REGION Network 12: Fittings - Cyle times measurement
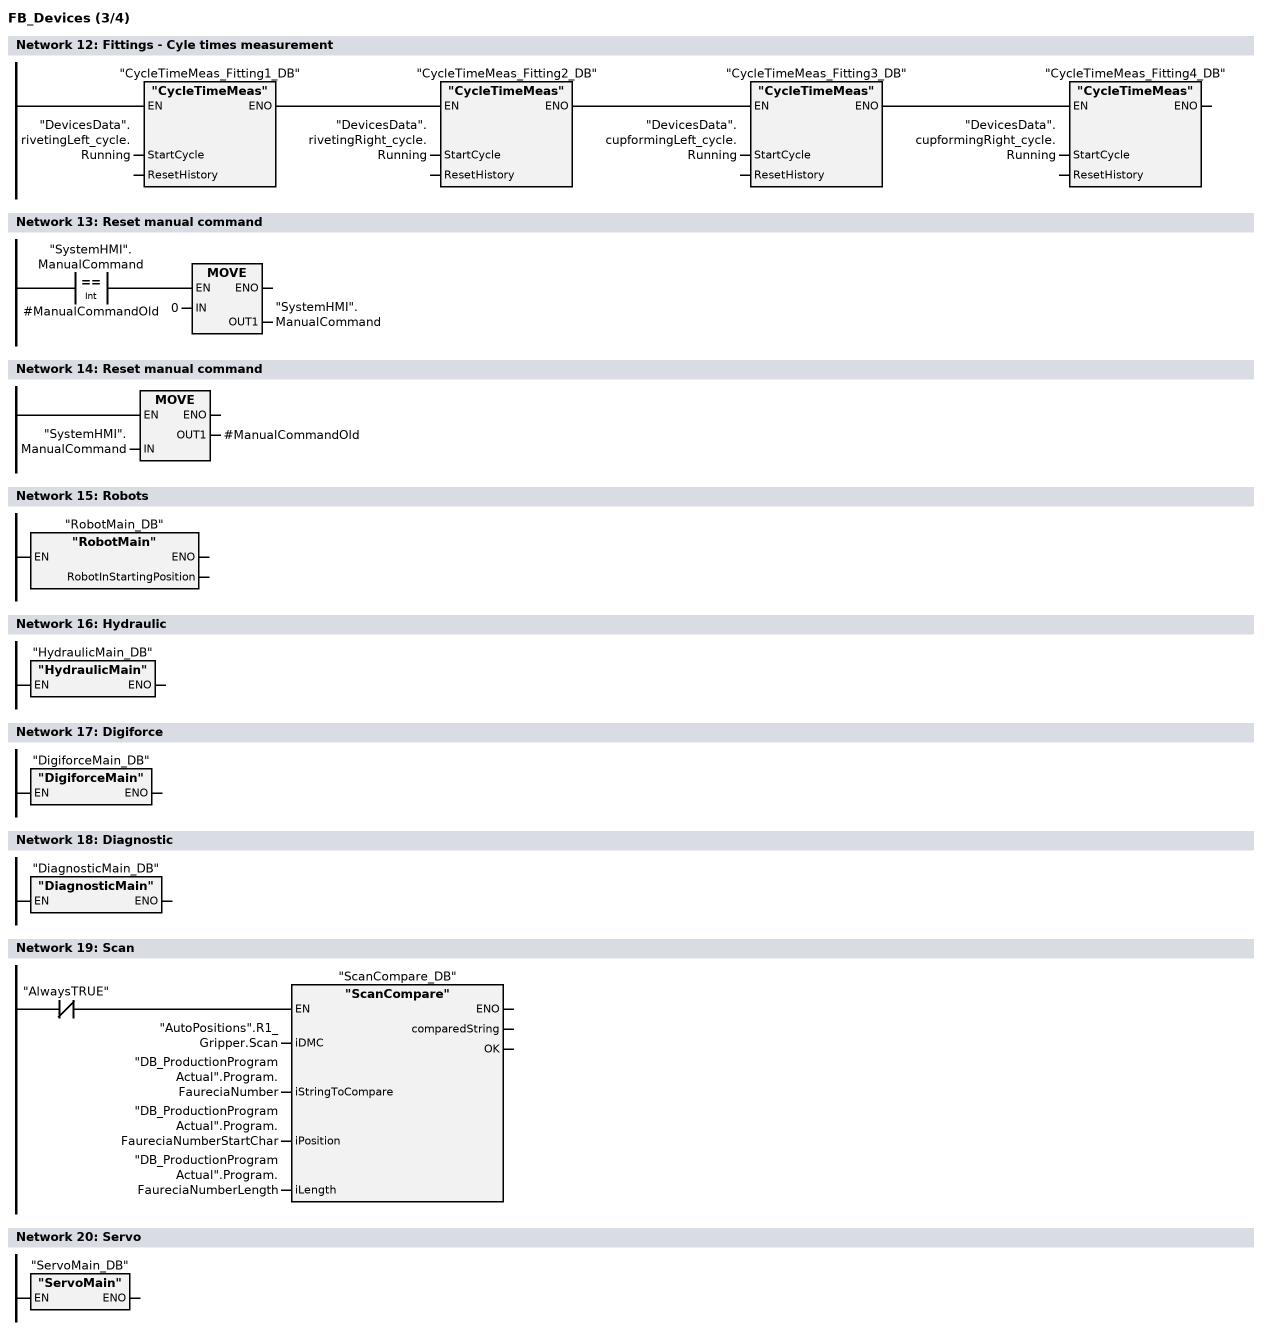
   RUNG wire#powerrail
      "CycleTimeMeas_Fitting1_DB"(StartCycle := "DevicesData".rivetingLeft_cycle.Running, ResetHistory :=)
      "CycleTimeMeas_Fitting2_DB"(StartCycle := "DevicesData".rivetingRight_cycle.Running, ResetHistory :=)
      "CycleTimeMeas_Fitting3_DB"(StartCycle := "DevicesData".cupformingLeft_cycle.Running, ResetHistory :=)
      "CycleTimeMeas_Fitting4_DB"(StartCycle := "DevicesData".cupformingRight_cycle.Running, ResetHistory :=)
   END_RUNG
   // the same network as SCL:
   "CycleTimeMeas_Fitting1_DB"(StartCycle := "DevicesData".rivetingLeft_cycle.Running, ENO => #_w1);   // "CycleTimeMeas"
   "CycleTimeMeas_Fitting2_DB"(EN := #_w1, StartCycle := "DevicesData".rivetingRight_cycle.Running, ENO => #_w2);   // "CycleTimeMeas"
   "CycleTimeMeas_Fitting3_DB"(EN := #_w2,   // "CycleTimeMeas"
                           StartCycle := "DevicesData".cupformingLeft_cycle.Running,
                           ENO => #_w3);
   IF #_w3 THEN
       "CycleTimeMeas_Fitting4_DB"(StartCycle := "DevicesData".cupformingRight_cycle.Running);   // "CycleTimeMeas"
   END_IF;
END_REGION

REGION Network 13: Reset manual command
   RUNG wire#powerrail
      { S7_Templates := "SrcType := Int" } EQ_Contact(in1 := "SystemHMI".ManualCommand, in2 := #ManualCommandOld)
      Move(in := 0, out1 => "SystemHMI".ManualCommand)
   END_RUNG
   // the same network as SCL:
   IF "SystemHMI".ManualCommand = #ManualCommandOld THEN "SystemHMI".ManualCommand := 0; END_IF;
END_REGION

REGION Network 14: Reset manual command
   RUNG wire#powerrail
      Move(in := "SystemHMI".ManualCommand, out1 => #ManualCommandOld)
   END_RUNG
   // the same network as SCL:
   #ManualCommandOld := "SystemHMI".ManualCommand;
END_REGION

REGION Network 15: Robots
   RUNG wire#powerrail
      "RobotMain_DB"(RobotInStartingPosition =>)
   END_RUNG
   // the same network as SCL:
   "RobotMain_DB"();   // "RobotMain"
END_REGION

REGION Network 16: Hydraulic
   RUNG wire#powerrail
      "HydraulicMain_DB"()
   END_RUNG
   // the same network as SCL:
   "HydraulicMain_DB"();   // "HydraulicMain"
END_REGION

REGION Network 17: Digiforce
   RUNG wire#powerrail
      "DigiforceMain_DB"()
   END_RUNG
   // the same network as SCL:
   "DigiforceMain_DB"();   // "DigiforceMain"
END_REGION

REGION Network 18: Diagnostic
   RUNG wire#powerrail
      "DiagnosticMain_DB"()
   END_RUNG
   // the same network as SCL:
   "DiagnosticMain_DB"();   // "DiagnosticMain"
END_REGION

REGION Network 19: Scan
   RUNG wire#powerrail
      I_Contact( "AlwaysTRUE" )
      "ScanCompare_DB"(iDMC := "AutoPositions".R1_Gripper.Scan, iStringToCompare := "DB_ProductionProgramActual".Program.FaureciaNumber, iPosition := "DB_ProductionProgramActual".Program.FaureciaNumberStartChar, iLength := "DB_ProductionProgramActual".Program.FaureciaNumberLength, comparedString =>, OK =>)
   END_RUNG
   // the same network as SCL:
   IF NOT "AlwaysTRUE" THEN
       "ScanCompare_DB"(iDMC := "AutoPositions".R1_Gripper.Scan,   // "ScanCompare"
                        iStringToCompare := "DB_ProductionProgramActual".Program.FaureciaNumber,
                        iPosition := "DB_ProductionProgramActual".Program.FaureciaNumberStartChar,
                        iLength := "DB_ProductionProgramActual".Program.FaureciaNumberLength);
   END_IF;
END_REGION

REGION Network 20: Servo
   RUNG wire#powerrail
      "ServoMain_DB"()
   END_RUNG
   // the same network as SCL:
   "ServoMain_DB"();   // "ServoMain"
END_REGION

REGION Network 21 (SCL): Friedrich1 R
   IF "HMIData".ManualCommand = 611 THEN
       "DevicesData".Friedrich1.Start := true;
   END_IF;

   #FriedrichUnit1_Instance(safetyOK := "safety_signals"."4L+",
                            iReady := "iRivetingReady1",
                            iZ1OK := "iRivetingZ1ok1",
                            iH1OK := "iRivetingH1ok1",
                            iH2OK := "iRivetingH2ok1",
                            iTimeOK := "iRivetingTimeOk1",
                            iNoAlarm := "iRivetingNoError1",
                            FriedrichNumber := 1,
                            Port := 39000,
                            IP1 := 192,
                            IP2 := 168,
                            IP3 := 16,
                            IP4 := 43,
                            ID := 2,
                            qStart => "qRiveting1Start",
                            qPrgbit4 => "qRiveting1Bit4",
                            qPrgbit3 => "qRiveting1Bit3",
                            qPrgbit2 => "qRiveting1Bit2",
                            qPrgbit1 => "qRiveting1Bit1",
                            qPrgbit0 => "qRiveting1Bit0",
                            RivetData := "DevicesData".Friedrich1);
   "qFriedrich1_setup_mode" := "DB_MainData".MachineMode <> 2 AND "DB_MainData".MachineMode <> 3;

   #Trig1(CLK:="DevicesData".Friedrich1.OK);
   #Trig2(CLK:="DevicesData".Friedrich1.NOK);
   "RivetingHistoryRight_DB"(iNewCycle := #Trig1.Q OR #Trig2.Q,
                             iData := "DevicesData".Friedrich1);

   #RivetingCycleRight_Instance(parameters := "DB_ProductionProgramActual".Program.Riveting_program_right,
                                basicPosition := "DevicesData".Friedrich1.Ready AND "DevicesData".Cylinders[MM340_RivetingUnitRight].InBp AND "DevicesData".Cylinders[MM344_RivetingSupportRight].InBp,
                                twoRivets := "DB_ProductionProgramActual".Program.Total_number_of_rivets_4,
                                MeasuredData1=>"AutoInfo".PartMeasuredData.RightRiveting1,
                                MeasuredData2=>"AutoInfo".PartMeasuredData.RightRiveting2,
                                riveter := "DevicesData".Friedrich1,
                                data := "DevicesData".rivetingRight_cycle,
                                cylinderSupport := "DevicesData".Cylinders[MM344_RivetingSupportRight],
                                cylinderShift := "DevicesData".Cylinders[MM340_RivetingUnitRight]);
END_REGION

REGION Network 22 (SCL): Friedrich2 L
   IF "HMIData".ManualCommand = 612 THEN
       "DevicesData".Friedrich2.Start := true;
   END_IF;
   #FriedrichUnit2_Instance(safetyOK := "safety_signals"."4L+",
                            iReady := "iRivetingReady2",
                            iZ1OK := "iRivetingZ1ok2",
                            iH1OK := "iRivetingH1ok2",
                            iH2OK := "iRivetingH2ok2",
                            iTimeOK := "iRivetingTimeOk2",
                            iNoAlarm := "iRivetingNoError2",
                            FriedrichNumber := 2,
                            Port := 39000,
                            IP1 := 192,
                            IP2 := 168,
                            IP3 := 16,
                            IP4 := 44,
                            ID := 3,
                            qStart => "qRiveting2Start",
                            qPrgbit4 => "qRiveting2Bit4",
                            qPrgbit3 => "qRiveting2Bit3",
                            qPrgbit2 => "qRiveting2Bit2",
                            qPrgbit1 => "qRiveting2Bit1",
                            qPrgbit0 => "qRiveting2Bit0",
                            RivetData := "DevicesData".Friedrich2);
   "qFriedrich2_setup_mode" := "DB_MainData".MachineMode <> 2 AND "DB_MainData".MachineMode <> 3;

   #Trig3(CLK:="DevicesData".Friedrich2.OK);
   #Trig4(CLK:="DevicesData".Friedrich2.NOK);
   "RivetingHistoryLeft_DB"(iNewCycle := #Trig3.Q OR #Trig4.Q,
                            iData := "DevicesData".Friedrich2);

   #RivetingCycleLeft_Instance(parameters := "DB_ProductionProgramActual".Program.Riveting_program_left,
                               basicPosition := "DevicesData".Friedrich2.Ready AND "DevicesData".Cylinders[MM342_RivetingUnitLeft].InBp AND "DevicesData".Cylinders[MM346_RivetingSupportLeft].InBp,
                               twoRivets := "DB_ProductionProgramActual".Program.Total_number_of_rivets_4,
                               MeasuredData1=>"AutoInfo".PartMeasuredData.LeftRiveting1,
                               MeasuredData2=>"AutoInfo".PartMeasuredData.LeftRiveting2,
                               riveter := "DevicesData".Friedrich2,
                               data := "DevicesData".rivetingLeft_cycle,
                               cylinderSupport := "DevicesData".Cylinders[MM346_RivetingSupportLeft],
                               cylinderShift := "DevicesData".Cylinders[MM342_RivetingUnitLeft]);

   REGION cycles handshake
       IF "SystemHMI".AutomaticMode THEN
           IF "DevicesData".cupformingLeft_cycle.Done AND "DevicesData".cupformingRight_cycle.Done THEN
               "DevicesData".rivetingLeft_cycle.ContinueFitting := TRUE;
               "DevicesData".rivetingRight_cycle.ContinueFitting := TRUE;
           END_IF;
       END_IF;
       "DevicesData".rivetingLeft_cycle.ContinueFitting := TRUE;
       "DevicesData".rivetingRight_cycle.ContinueFitting := TRUE;

       IF "SystemHMI".ManualMode THEN
           "DevicesData".rivetingLeft_cycle.ContinueFitting := true;
           "DevicesData".rivetingRight_cycle.ContinueFitting := true;
       END_IF;
   END_REGION
END_REGION

REGION Network 23
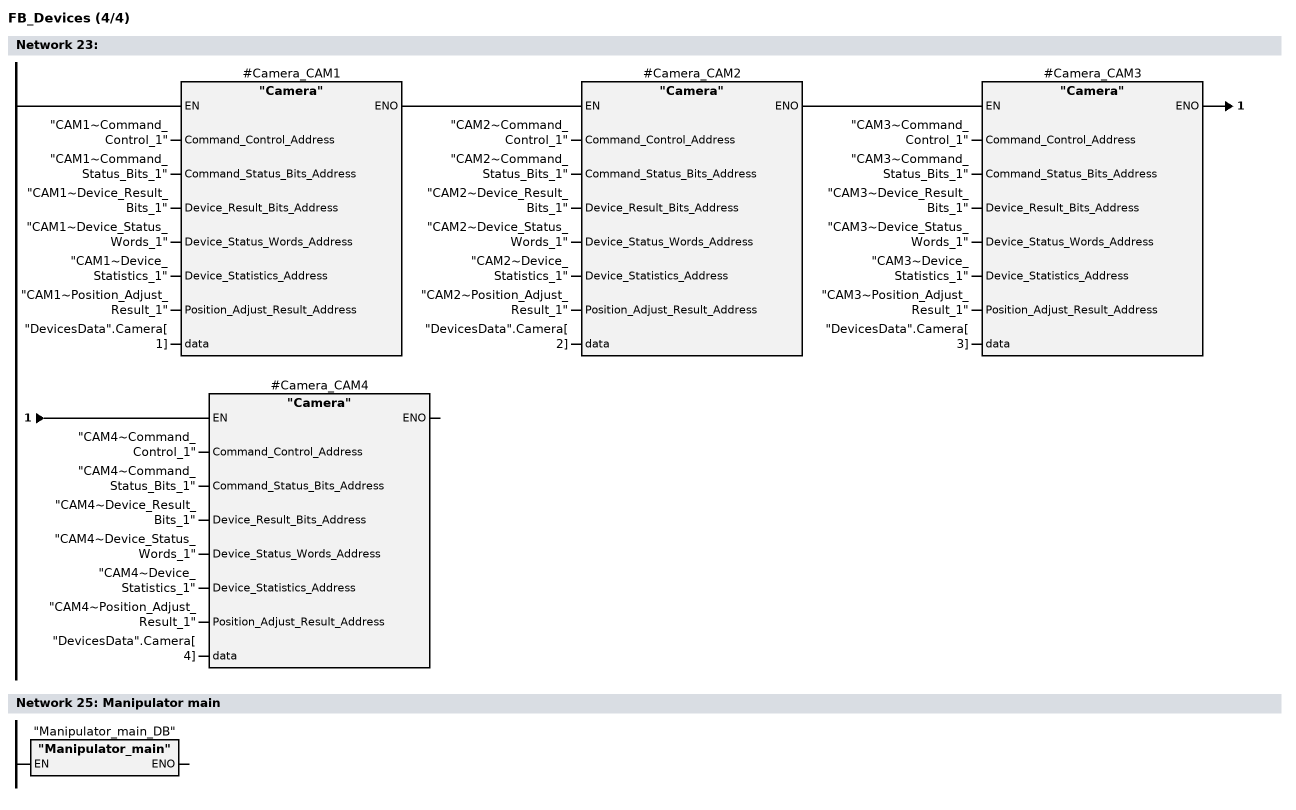
   RUNG wire#powerrail
      #Camera_CAM1(Command_Control_Address := "CAM1~Command_Control_1", Command_Status_Bits_Address := "CAM1~Command_Status_Bits_1", Device_Result_Bits_Address := "CAM1~Device_Result_Bits_1", Device_Status_Words_Address := "CAM1~Device_Status_Words_1", Device_Statistics_Address := "CAM1~Device_Statistics_1", Position_Adjust_Result_Address := "CAM1~Position_Adjust_Result_1", data := "DevicesData".Camera[1])
      #Camera_CAM2(Command_Control_Address := "CAM2~Command_Control_1", Command_Status_Bits_Address := "CAM2~Command_Status_Bits_1", Device_Result_Bits_Address := "CAM2~Device_Result_Bits_1", Device_Status_Words_Address := "CAM2~Device_Status_Words_1", Device_Statistics_Address := "CAM2~Device_Statistics_1", Position_Adjust_Result_Address := "CAM2~Position_Adjust_Result_1", data := "DevicesData".Camera[2])
      #Camera_CAM3(Command_Control_Address := "CAM3~Command_Control_1", Command_Status_Bits_Address := "CAM3~Command_Status_Bits_1", Device_Result_Bits_Address := "CAM3~Device_Result_Bits_1", Device_Status_Words_Address := "CAM3~Device_Status_Words_1", Device_Statistics_Address := "CAM3~Device_Statistics_1", Position_Adjust_Result_Address := "CAM3~Position_Adjust_Result_1", data := "DevicesData".Camera[3])
      #Camera_CAM4(Command_Control_Address := "CAM4~Command_Control_1", Command_Status_Bits_Address := "CAM4~Command_Status_Bits_1", Device_Result_Bits_Address := "CAM4~Device_Result_Bits_1", Device_Status_Words_Address := "CAM4~Device_Status_Words_1", Device_Statistics_Address := "CAM4~Device_Statistics_1", Position_Adjust_Result_Address := "CAM4~Position_Adjust_Result_1", data := "DevicesData".Camera[4])
   END_RUNG
   // the same network as SCL:
   #Camera_CAM1(Command_Control_Address := "CAM1~Command_Control_1",   // "Camera"
                Command_Status_Bits_Address := "CAM1~Command_Status_Bits_1",
                Device_Result_Bits_Address := "CAM1~Device_Result_Bits_1",
                Device_Status_Words_Address := "CAM1~Device_Status_Words_1",
                Device_Statistics_Address := "CAM1~Device_Statistics_1",
                Position_Adjust_Result_Address := "CAM1~Position_Adjust_Result_1",
                data := "DevicesData".Camera[1],
                ENO => #_w1);
   #Camera_CAM2(EN := #_w1,   // "Camera"
                Command_Control_Address := "CAM2~Command_Control_1",
                Command_Status_Bits_Address := "CAM2~Command_Status_Bits_1",
                Device_Result_Bits_Address := "CAM2~Device_Result_Bits_1",
                Device_Status_Words_Address := "CAM2~Device_Status_Words_1",
                Device_Statistics_Address := "CAM2~Device_Statistics_1",
                Position_Adjust_Result_Address := "CAM2~Position_Adjust_Result_1",
                data := "DevicesData".Camera[2],
                ENO => #_w2);
   #Camera_CAM3(EN := #_w2,   // "Camera"
                Command_Control_Address := "CAM3~Command_Control_1",
                Command_Status_Bits_Address := "CAM3~Command_Status_Bits_1",
                Device_Result_Bits_Address := "CAM3~Device_Result_Bits_1",
                Device_Status_Words_Address := "CAM3~Device_Status_Words_1",
                Device_Statistics_Address := "CAM3~Device_Statistics_1",
                Position_Adjust_Result_Address := "CAM3~Position_Adjust_Result_1",
                data := "DevicesData".Camera[3],
                ENO => #_w3);
   IF #_w3 THEN
       #Camera_CAM4(Command_Control_Address := "CAM4~Command_Control_1",   // "Camera"
                    Command_Status_Bits_Address := "CAM4~Command_Status_Bits_1",
                    Device_Result_Bits_Address := "CAM4~Device_Result_Bits_1",
                    Device_Status_Words_Address := "CAM4~Device_Status_Words_1",
                    Device_Statistics_Address := "CAM4~Device_Statistics_1",
                    Position_Adjust_Result_Address := "CAM4~Position_Adjust_Result_1",
                    data := "DevicesData".Camera[4]);
   END_IF;
END_REGION

REGION Network 24 (SCL)
   "DevicesData".Camera[1].ProgramNumber := USINT_TO_SINT("DB_ProductionProgramActual".Program.Camera_program[1]);
   "DevicesData".Camera[2].ProgramNumber := USINT_TO_SINT("DB_ProductionProgramActual".Program.Camera_program[2]);
   "DevicesData".Camera[3].ProgramNumber := USINT_TO_SINT("DB_ProductionProgramActual".Program.Camera_program[3]);
   "DevicesData".Camera[4].ProgramNumber := USINT_TO_SINT("DB_ProductionProgramActual".Program.Camera_program[4]);
END_REGION

REGION Network 25: Manipulator main
   RUNG wire#powerrail
      "Manipulator_main_DB"()
   END_RUNG
   // the same network as SCL:
   "Manipulator_main_DB"();   // "Manipulator_main"
END_REGION

REGION Network 26: Readers
END_REGION
END_FUNCTION_BLOCK

FUNCTION_BLOCK "CylindersMain"
{ S7_Optimized_Access := 'TRUE' }
VERSION : 0.1
   VAR 
      res : Bool;
   END_VAR


BEGIN
	
	"CylinderGeneratedCalls_DB"();
	
	"CylinderCollisions"();
	
	"CylindersHMIMessage"(CylinderNumber=>"CylindersHMI".CylinderInfoHMI,
	                      CylinderAction=>"CylindersHMI".CylinderInfoHMIAction);
	
END_FUNCTION_BLOCK

FUNCTION_BLOCK "FB_TurnTable"   // FB3600, LAD
{ S7_Optimized_Access := 'TRUE' }
VERSION : 0.1
// stored: AutoNumber false, IsIECCheckEnabled false, IsRetainMemResEnabled false, MemoryReserve 100, SetENOAutomatically false, UDAEnableTagReadback false
   VAR_INPUT
      iTurnTableInputs : Word;
      iPower : Bool;
      iSafety : Bool;
      iReset : Bool;
      iErrorReset : Bool;
      iManualMode : Bool;
      iAutomaticMode : Bool;
      iTurnTableInSafetyPosition : Bool;
   END_VAR
   VAR_OUTPUT
      qTurnTableOutputs : Word;
      qeCommunication : Bool;
      qeTurnTablePosition : Bool;
      qeTurnTableSafetyPosition : Bool;
      qeTimeout : Bool;
      qePositionRunOver : Bool;
      qeSafety : Bool;
      qeSumError : Bool;
      qeSumWarning : Bool;
   END_VAR
   VAR_IN_OUT
      iqTurnTable : "UDT_TurnTable";
   END_VAR
   VAR
      Edges : Struct
         Enabled : Bool;
         IndexerInPosition : Bool;
      END_STRUCT;
      TONs : Struct
         tDelayCommunication : TON_TIME;
         tDelayPositionError { S7_SetPoint := 'True'} : TON_TIME;
         tDelayErrorReset { S7_SetPoint := 'True'} : TON_TIME;
      END_STRUCT;
   END_VAR
   VAR RETAIN
      RetentiveData : Struct
         LastDirection : Bool;
      END_STRUCT;
   END_VAR
   VAR
      Commands : "UDT_TurnTableCommands";
   END_VAR
   VAR_TEMP
      mode_status : Struct
         manual_mode : Bool;
         automatic_mode : Bool;
         mode_active : Bool;
      END_STRUCT;
      bit : Bool;
      error : Bool;
      ready_to_cw : Bool;
      ready_to_ccw : Bool;
      ready_to_jog : Bool;
      ready_to_start : Bool;
   END_VAR
   VAR_TEMP   // added for the SCL form of the ladder/FBD networks
      _w1 : Bool;
      _w2 : Bool;
      _w3 : Bool;
   END_VAR
BEGIN

REGION Network 1: Read inputs
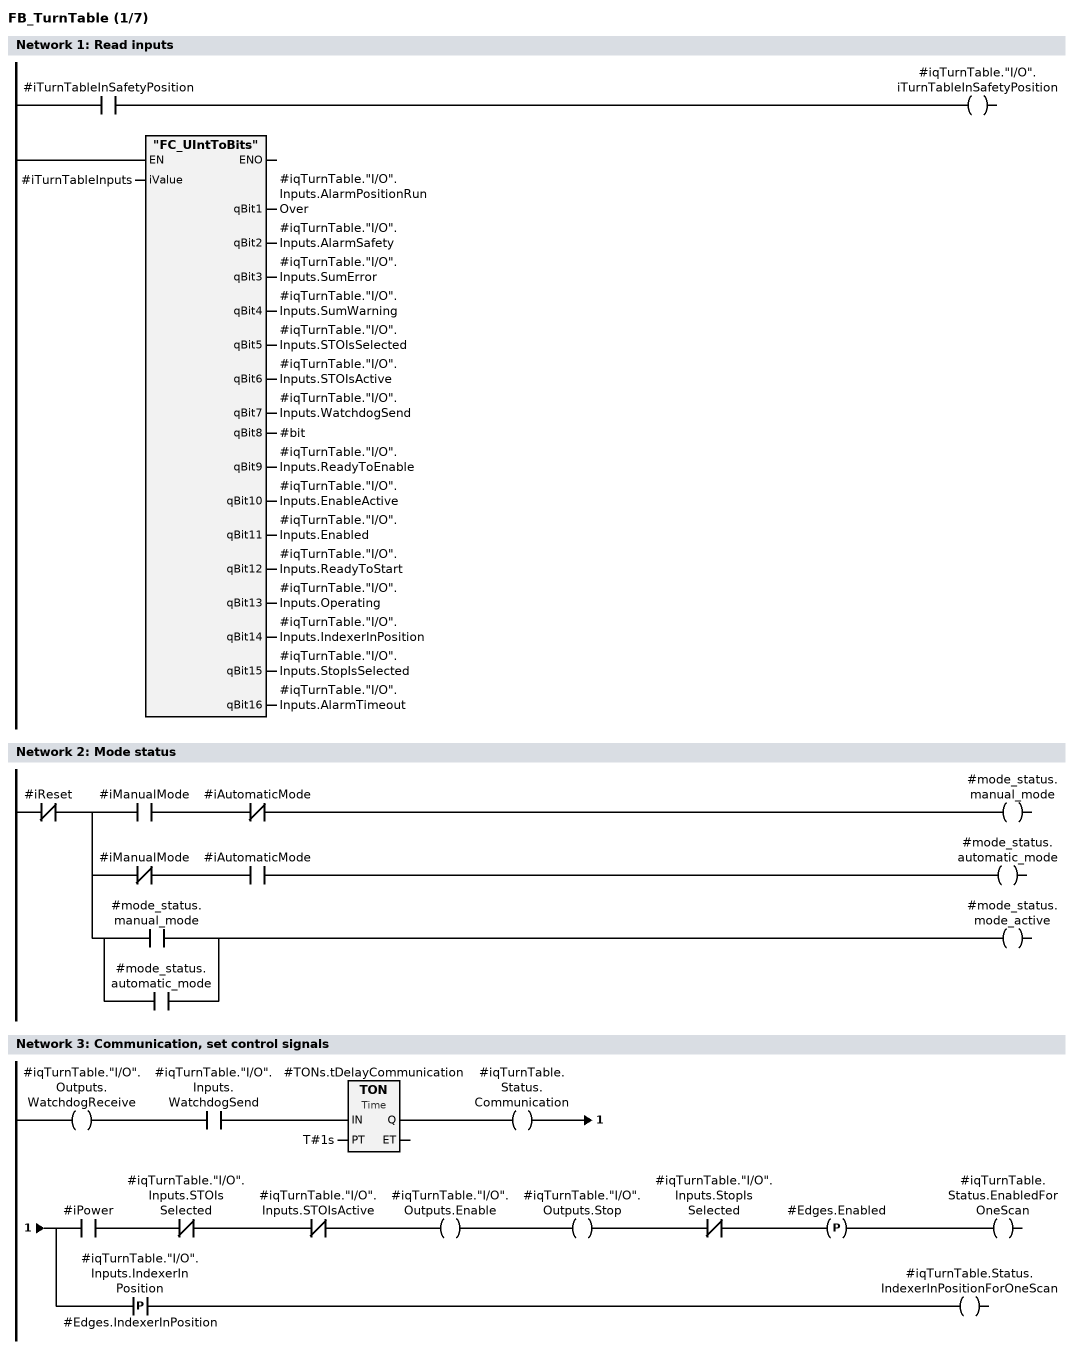
   RUNG wire#powerrail
      Contact( #iTurnTableInSafetyPosition )
      Coil( #iqTurnTable."I/O".iTurnTableInSafetyPosition )
   END_RUNG
   RUNG wire#powerrail
      "FC_UIntToBits"(iValue := #iTurnTableInputs, qBit1 => #iqTurnTable."I/O".Inputs.AlarmPositionRunOver, qBit2 => #iqTurnTable."I/O".Inputs.AlarmSafety, qBit3 => #iqTurnTable."I/O".Inputs.SumError, qBit4 => #iqTurnTable."I/O".Inputs.SumWarning, qBit5 => #iqTurnTable."I/O".Inputs.STOIsSelected, qBit6 => #iqTurnTable."I/O".Inputs.STOIsActive, qBit7 => #iqTurnTable."I/O".Inputs.WatchdogSend, qBit8 => #bit, qBit9 => #iqTurnTable."I/O".Inputs.ReadyToEnable, qBit10 => #iqTurnTable."I/O".Inputs.EnableActive, qBit11 => #iqTurnTable."I/O".Inputs.Enabled, qBit12 => #iqTurnTable."I/O".Inputs.ReadyToStart, qBit13 => #iqTurnTable."I/O".Inputs.Operating, qBit14 => #iqTurnTable."I/O".Inputs.IndexerInPosition, qBit15 => #iqTurnTable."I/O".Inputs.StopIsSelected, qBit16 => #iqTurnTable."I/O".Inputs.AlarmTimeout)
   END_RUNG
   // the same network as SCL:
   #iqTurnTable."I/O".iTurnTableInSafetyPosition := #iTurnTableInSafetyPosition;
   "FC_UIntToBits"(iValue := #iTurnTableInputs,
                   qBit1 => #iqTurnTable."I/O".Inputs.AlarmPositionRunOver,
                   qBit2 => #iqTurnTable."I/O".Inputs.AlarmSafety,
                   qBit3 => #iqTurnTable."I/O".Inputs.SumError,
                   qBit4 => #iqTurnTable."I/O".Inputs.SumWarning,
                   qBit5 => #iqTurnTable."I/O".Inputs.STOIsSelected,
                   qBit6 => #iqTurnTable."I/O".Inputs.STOIsActive,
                   qBit7 => #iqTurnTable."I/O".Inputs.WatchdogSend,
                   qBit8 => #bit,
                   qBit9 => #iqTurnTable."I/O".Inputs.ReadyToEnable,
                   qBit10 => #iqTurnTable."I/O".Inputs.EnableActive,
                   qBit11 => #iqTurnTable."I/O".Inputs.Enabled,
                   qBit12 => #iqTurnTable."I/O".Inputs.ReadyToStart,
                   qBit13 => #iqTurnTable."I/O".Inputs.Operating,
                   qBit14 => #iqTurnTable."I/O".Inputs.IndexerInPosition,
                   qBit15 => #iqTurnTable."I/O".Inputs.StopIsSelected,
                   qBit16 => #iqTurnTable."I/O".Inputs.AlarmTimeout);
END_REGION

REGION Network 2: Mode status
   RUNG wire#powerrail
      I_Contact( #iReset )
      wire#w1
      Contact( #iManualMode )
      I_Contact( #iAutomaticMode )
      Coil( #mode_status.manual_mode )
   END_RUNG
   RUNG wire#w1
      I_Contact( #iManualMode )
      Contact( #iAutomaticMode )
      Coil( #mode_status.automatic_mode )
   END_RUNG
   RUNG wire#w1
      Contact( #mode_status.manual_mode )
      wire#w2
      Coil( #mode_status.mode_active )
   END_RUNG
   RUNG wire#w1
      Contact( #mode_status.automatic_mode )
   END_RUNG wire#w2
   // the same network as SCL:
   #mode_status.manual_mode := NOT #iReset AND #iManualMode AND NOT #iAutomaticMode;
   #mode_status.automatic_mode := NOT #iReset AND NOT #iManualMode AND #iAutomaticMode;
   #mode_status.mode_active := NOT #iReset AND (#mode_status.manual_mode OR #mode_status.automatic_mode);
END_REGION

REGION Network 3: Communication, set control signals
   RUNG wire#powerrail
      Coil( #iqTurnTable."I/O".Outputs.WatchdogReceive )
      Contact( #iqTurnTable."I/O".Inputs.WatchdogSend )
      { S7_Templates := "time_type := Time" } #TONs.tDelayCommunication.TON(pt := T#1s, et =>)
      Coil( #iqTurnTable.Status.Communication )
      wire#w1
      Contact( #iPower )
      I_Contact( #iqTurnTable."I/O".Inputs.STOIsSelected )
      I_Contact( #iqTurnTable."I/O".Inputs.STOIsActive )
      Coil( #iqTurnTable."I/O".Outputs.Enable )
      Coil( #iqTurnTable."I/O".Outputs.Stop )
      I_Contact( #iqTurnTable."I/O".Inputs.StopIsSelected )
      P_Trig( #Edges.Enabled )
      Coil( #iqTurnTable.Status.EnabledForOneScan )
   END_RUNG
   RUNG wire#w1
      P_Contact(operand := #iqTurnTable."I/O".Inputs.IndexerInPosition, bit := #Edges.IndexerInPosition)
      Coil( #iqTurnTable.Status.IndexerInPositionForOneScan )
   END_RUNG
   // the same network as SCL:
   #iqTurnTable."I/O".Outputs.WatchdogReceive := TRUE;
   #TONs.tDelayCommunication.TON(IN := #iqTurnTable."I/O".Inputs.WatchdogSend, PT := T#1s);
   #iqTurnTable.Status.Communication := #TONs.tDelayCommunication.Q;
   #iqTurnTable."I/O".Outputs.Enable := #TONs.tDelayCommunication.Q AND #iPower AND NOT #iqTurnTable."I/O".Inputs.STOIsSelected AND NOT #iqTurnTable."I/O".Inputs.STOIsActive;
   #iqTurnTable."I/O".Outputs.Stop := #iqTurnTable."I/O".Outputs.Enable;
   #_w1 := #iqTurnTable."I/O".Outputs.Enable AND NOT #iqTurnTable."I/O".Inputs.StopIsSelected;
   #_w2 := #_w1 AND NOT #Edges.Enabled;   // rising edge
   #Edges.Enabled := #_w1;
   #iqTurnTable.Status.EnabledForOneScan := #_w2;
   #_w3 := #TONs.tDelayCommunication.Q AND #iqTurnTable."I/O".Inputs.IndexerInPosition AND NOT #Edges.IndexerInPosition;   // rising edge of #iqTurnTable."I/O".Inputs.IndexerInPosition
   #Edges.IndexerInPosition := #iqTurnTable."I/O".Inputs.IndexerInPosition;
   #iqTurnTable.Status.IndexerInPositionForOneScan := #_w3;
END_REGION

REGION Network 4: Errors
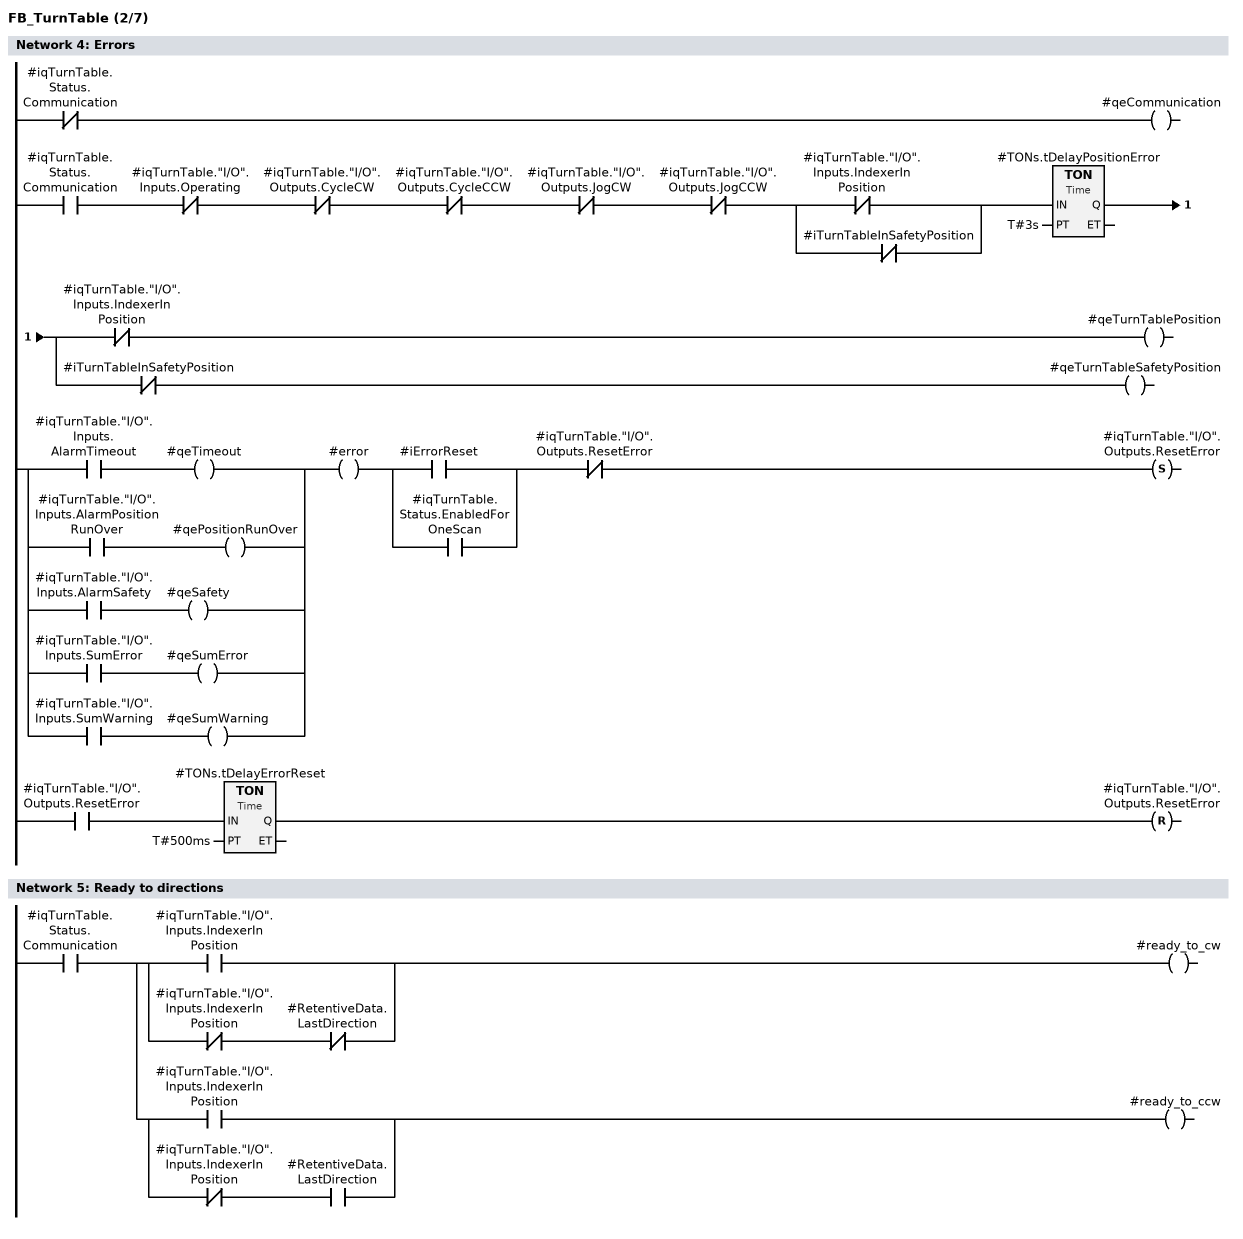
   RUNG wire#powerrail
      I_Contact( #iqTurnTable.Status.Communication )
      Coil( #qeCommunication )
   END_RUNG
   RUNG wire#powerrail
      Contact( #iqTurnTable.Status.Communication )
      I_Contact( #iqTurnTable."I/O".Inputs.Operating )
      I_Contact( #iqTurnTable."I/O".Outputs.CycleCW )
      I_Contact( #iqTurnTable."I/O".Outputs.CycleCCW )
      I_Contact( #iqTurnTable."I/O".Outputs.JogCW )
      I_Contact( #iqTurnTable."I/O".Outputs.JogCCW )
      wire#w1
      I_Contact( #iqTurnTable."I/O".Inputs.IndexerInPosition )
      wire#w2
      { S7_Templates := "time_type := Time" } #TONs.tDelayPositionError.TON(pt := T#3s, et =>)
      wire#w3
      I_Contact( #iqTurnTable."I/O".Inputs.IndexerInPosition )
      Coil( #qeTurnTablePosition )
   END_RUNG
   RUNG wire#w1
      I_Contact( #iTurnTableInSafetyPosition )
   END_RUNG wire#w2
   RUNG wire#w3
      I_Contact( #iTurnTableInSafetyPosition )
      Coil( #qeTurnTableSafetyPosition )
   END_RUNG
   RUNG wire#powerrail
      Contact( #iqTurnTable."I/O".Inputs.AlarmTimeout )
      Coil( #qeTimeout )
      wire#w4
      Coil( #error )
      wire#w5
      Contact( #iErrorReset )
      wire#w6
      I_Contact( #iqTurnTable."I/O".Outputs.ResetError )
      S_Coil( #iqTurnTable."I/O".Outputs.ResetError )
   END_RUNG
   RUNG wire#powerrail
      Contact( #iqTurnTable."I/O".Inputs.AlarmPositionRunOver )
      Coil( #qePositionRunOver )
   END_RUNG wire#w4
   RUNG wire#powerrail
      Contact( #iqTurnTable."I/O".Inputs.AlarmSafety )
      Coil( #qeSafety )
   END_RUNG wire#w4
   RUNG wire#powerrail
      Contact( #iqTurnTable."I/O".Inputs.SumError )
      Coil( #qeSumError )
   END_RUNG wire#w4
   RUNG wire#powerrail
      Contact( #iqTurnTable."I/O".Inputs.SumWarning )
      Coil( #qeSumWarning )
   END_RUNG wire#w4
   RUNG wire#w5
      Contact( #iqTurnTable.Status.EnabledForOneScan )
   END_RUNG wire#w6
   RUNG wire#powerrail
      Contact( #iqTurnTable."I/O".Outputs.ResetError )
      { S7_Templates := "time_type := Time" } #TONs.tDelayErrorReset.TON(pt := T#500ms, et =>)
      R_Coil( #iqTurnTable."I/O".Outputs.ResetError )
   END_RUNG
   // the same network as SCL:
   #qeCommunication := NOT #iqTurnTable.Status.Communication;
   #TONs.tDelayPositionError.TON(IN := #iqTurnTable.Status.Communication AND NOT #iqTurnTable."I/O".Inputs.Operating AND NOT #iqTurnTable."I/O".Outputs.CycleCW AND NOT #iqTurnTable."I/O".Outputs.CycleCCW AND NOT #iqTurnTable."I/O".Outputs.JogCW AND NOT #iqTurnTable."I/O".Outputs.JogCCW AND (NOT #iqTurnTable."I/O".Inputs.IndexerInPosition OR NOT #iTurnTableInSafetyPosition),
                           PT := T#3s);
   #qeTurnTablePosition := #TONs.tDelayPositionError.Q AND NOT #iqTurnTable."I/O".Inputs.IndexerInPosition;
   #qeTurnTableSafetyPosition := #TONs.tDelayPositionError.Q AND NOT #iTurnTableInSafetyPosition;
   #qeTimeout := #iqTurnTable."I/O".Inputs.AlarmTimeout;
   #qePositionRunOver := #iqTurnTable."I/O".Inputs.AlarmPositionRunOver;
   #qeSafety := #iqTurnTable."I/O".Inputs.AlarmSafety;
   #qeSumError := #iqTurnTable."I/O".Inputs.SumError;
   #qeSumWarning := #iqTurnTable."I/O".Inputs.SumWarning;
   #error := #iqTurnTable."I/O".Inputs.AlarmTimeout OR #iqTurnTable."I/O".Inputs.AlarmPositionRunOver OR #iqTurnTable."I/O".Inputs.AlarmSafety OR #iqTurnTable."I/O".Inputs.SumError OR #iqTurnTable."I/O".Inputs.SumWarning;
   IF #error AND (#iErrorReset OR #iqTurnTable.Status.EnabledForOneScan) AND NOT #iqTurnTable."I/O".Outputs.ResetError THEN
       #iqTurnTable."I/O".Outputs.ResetError := TRUE;
   END_IF;
   #TONs.tDelayErrorReset.TON(IN := #iqTurnTable."I/O".Outputs.ResetError, PT := T#500ms);
   IF #TONs.tDelayErrorReset.Q THEN #iqTurnTable."I/O".Outputs.ResetError := FALSE; END_IF;
END_REGION

REGION Network 5: Ready to directions
   RUNG wire#powerrail
      Contact( #iqTurnTable.Status.Communication )
      wire#w1
      Contact( #iqTurnTable."I/O".Inputs.IndexerInPosition )
      wire#w2
      Coil( #ready_to_cw )
   END_RUNG
   RUNG wire#w1
      I_Contact( #iqTurnTable."I/O".Inputs.IndexerInPosition )
      I_Contact( #RetentiveData.LastDirection )
   END_RUNG wire#w2
   RUNG wire#w1
      Contact( #iqTurnTable."I/O".Inputs.IndexerInPosition )
      wire#w3
      Coil( #ready_to_ccw )
   END_RUNG
   RUNG wire#w1
      I_Contact( #iqTurnTable."I/O".Inputs.IndexerInPosition )
      Contact( #RetentiveData.LastDirection )
   END_RUNG wire#w3
   // the same network as SCL:
   #ready_to_cw := #iqTurnTable.Status.Communication AND (#iqTurnTable."I/O".Inputs.IndexerInPosition OR (NOT #iqTurnTable."I/O".Inputs.IndexerInPosition AND NOT #RetentiveData.LastDirection));
   #ready_to_ccw := #iqTurnTable.Status.Communication AND (#iqTurnTable."I/O".Inputs.IndexerInPosition OR (NOT #iqTurnTable."I/O".Inputs.IndexerInPosition AND #RetentiveData.LastDirection));
END_REGION

REGION Network 6: Ready to jog
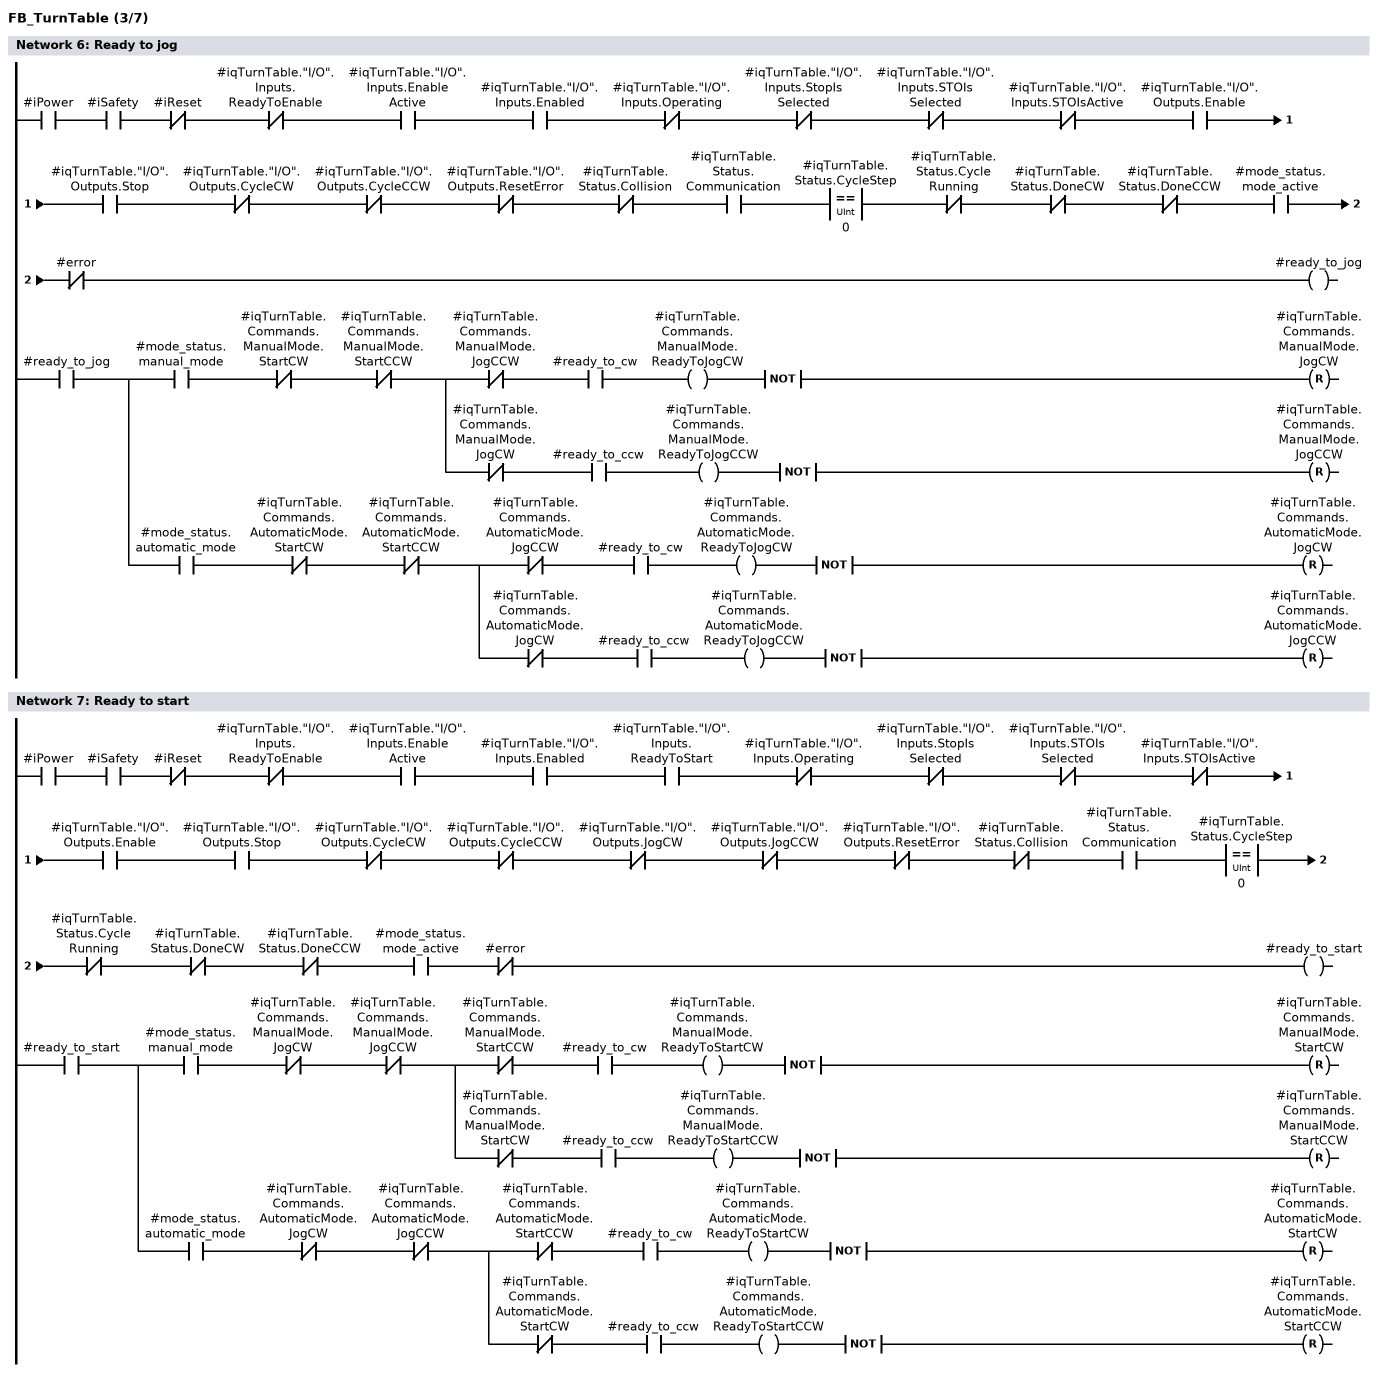
   RUNG wire#powerrail
      Contact( #iPower )
      Contact( #iSafety )
      I_Contact( #iReset )
      I_Contact( #iqTurnTable."I/O".Inputs.ReadyToEnable )
      Contact( #iqTurnTable."I/O".Inputs.EnableActive )
      Contact( #iqTurnTable."I/O".Inputs.Enabled )
      I_Contact( #iqTurnTable."I/O".Inputs.Operating )
      I_Contact( #iqTurnTable."I/O".Inputs.StopIsSelected )
      I_Contact( #iqTurnTable."I/O".Inputs.STOIsSelected )
      I_Contact( #iqTurnTable."I/O".Inputs.STOIsActive )
      Contact( #iqTurnTable."I/O".Outputs.Enable )
      Contact( #iqTurnTable."I/O".Outputs.Stop )
      I_Contact( #iqTurnTable."I/O".Outputs.CycleCW )
      I_Contact( #iqTurnTable."I/O".Outputs.CycleCCW )
      I_Contact( #iqTurnTable."I/O".Outputs.ResetError )
      I_Contact( #iqTurnTable.Status.Collision )
      Contact( #iqTurnTable.Status.Communication )
      { S7_Templates := "SrcType := UInt" } EQ_Contact(in1 := #iqTurnTable.Status.CycleStep, in2 := 0)
      I_Contact( #iqTurnTable.Status.CycleRunning )
      I_Contact( #iqTurnTable.Status.DoneCW )
      I_Contact( #iqTurnTable.Status.DoneCCW )
      Contact( #mode_status.mode_active )
      I_Contact( #error )
      Coil( #ready_to_jog )
   END_RUNG
   RUNG wire#powerrail
      Contact( #ready_to_jog )
      wire#w1
      Contact( #mode_status.manual_mode )
      I_Contact( #iqTurnTable.Commands.ManualMode.StartCW )
      I_Contact( #iqTurnTable.Commands.ManualMode.StartCCW )
      wire#w2
      I_Contact( #iqTurnTable.Commands.ManualMode.JogCCW )
      Contact( #ready_to_cw )
      Coil( #iqTurnTable.Commands.ManualMode.ReadyToJogCW )
      Not()
      R_Coil( #iqTurnTable.Commands.ManualMode.JogCW )
   END_RUNG
   RUNG wire#w2
      I_Contact( #iqTurnTable.Commands.ManualMode.JogCW )
      Contact( #ready_to_ccw )
      Coil( #iqTurnTable.Commands.ManualMode.ReadyToJogCCW )
      Not()
      R_Coil( #iqTurnTable.Commands.ManualMode.JogCCW )
   END_RUNG
   RUNG wire#w1
      Contact( #mode_status.automatic_mode )
      I_Contact( #iqTurnTable.Commands.AutomaticMode.StartCW )
      I_Contact( #iqTurnTable.Commands.AutomaticMode.StartCCW )
      wire#w3
      I_Contact( #iqTurnTable.Commands.AutomaticMode.JogCCW )
      Contact( #ready_to_cw )
      Coil( #iqTurnTable.Commands.AutomaticMode.ReadyToJogCW )
      Not()
      R_Coil( #iqTurnTable.Commands.AutomaticMode.JogCW )
   END_RUNG
   RUNG wire#w3
      I_Contact( #iqTurnTable.Commands.AutomaticMode.JogCW )
      Contact( #ready_to_ccw )
      Coil( #iqTurnTable.Commands.AutomaticMode.ReadyToJogCCW )
      Not()
      R_Coil( #iqTurnTable.Commands.AutomaticMode.JogCCW )
   END_RUNG
   // the same network as SCL:
   #ready_to_jog := #iPower AND #iSafety AND NOT #iReset AND NOT #iqTurnTable."I/O".Inputs.ReadyToEnable AND #iqTurnTable."I/O".Inputs.EnableActive AND #iqTurnTable."I/O".Inputs.Enabled AND NOT #iqTurnTable."I/O".Inputs.Operating AND NOT #iqTurnTable."I/O".Inputs.StopIsSelected AND NOT #iqTurnTable."I/O".Inputs.STOIsSelected AND NOT #iqTurnTable."I/O".Inputs.STOIsActive AND #iqTurnTable."I/O".Outputs.Enable AND #iqTurnTable."I/O".Outputs.Stop AND NOT #iqTurnTable."I/O".Outputs.CycleCW AND NOT #iqTurnTable."I/O".Outputs.CycleCCW AND NOT #iqTurnTable."I/O".Outputs.ResetError AND NOT #iqTurnTable.Status.Collision AND #iqTurnTable.Status.Communication AND (#iqTurnTable.Status.CycleStep = 0) AND NOT #iqTurnTable.Status.CycleRunning AND NOT #iqTurnTable.Status.DoneCW AND NOT #iqTurnTable.Status.DoneCCW AND #mode_status.mode_active AND NOT #error;
   #_w1 := #ready_to_jog AND #mode_status.manual_mode AND NOT #iqTurnTable.Commands.ManualMode.StartCW AND NOT #iqTurnTable.Commands.ManualMode.StartCCW;
   #iqTurnTable.Commands.ManualMode.ReadyToJogCW := #_w1 AND NOT #iqTurnTable.Commands.ManualMode.JogCCW AND #ready_to_cw;
   IF NOT #iqTurnTable.Commands.ManualMode.ReadyToJogCW THEN
       #iqTurnTable.Commands.ManualMode.JogCW := FALSE;
   END_IF;
   #iqTurnTable.Commands.ManualMode.ReadyToJogCCW := #_w1 AND NOT #iqTurnTable.Commands.ManualMode.JogCW AND #ready_to_ccw;
   IF NOT #iqTurnTable.Commands.ManualMode.ReadyToJogCCW THEN
       #iqTurnTable.Commands.ManualMode.JogCCW := FALSE;
   END_IF;
   #_w2 := #ready_to_jog AND #mode_status.automatic_mode AND NOT #iqTurnTable.Commands.AutomaticMode.StartCW AND NOT #iqTurnTable.Commands.AutomaticMode.StartCCW;
   #iqTurnTable.Commands.AutomaticMode.ReadyToJogCW := #_w2 AND NOT #iqTurnTable.Commands.AutomaticMode.JogCCW AND #ready_to_cw;
   IF NOT #iqTurnTable.Commands.AutomaticMode.ReadyToJogCW THEN
       #iqTurnTable.Commands.AutomaticMode.JogCW := FALSE;
   END_IF;
   #iqTurnTable.Commands.AutomaticMode.ReadyToJogCCW := #_w2 AND NOT #iqTurnTable.Commands.AutomaticMode.JogCW AND #ready_to_ccw;
   IF NOT #iqTurnTable.Commands.AutomaticMode.ReadyToJogCCW THEN
       #iqTurnTable.Commands.AutomaticMode.JogCCW := FALSE;
   END_IF;
END_REGION

REGION Network 7: Ready to start
   RUNG wire#powerrail
      Contact( #iPower )
      Contact( #iSafety )
      I_Contact( #iReset )
      I_Contact( #iqTurnTable."I/O".Inputs.ReadyToEnable )
      Contact( #iqTurnTable."I/O".Inputs.EnableActive )
      Contact( #iqTurnTable."I/O".Inputs.Enabled )
      Contact( #iqTurnTable."I/O".Inputs.ReadyToStart )
      I_Contact( #iqTurnTable."I/O".Inputs.Operating )
      I_Contact( #iqTurnTable."I/O".Inputs.StopIsSelected )
      I_Contact( #iqTurnTable."I/O".Inputs.STOIsSelected )
      I_Contact( #iqTurnTable."I/O".Inputs.STOIsActive )
      Contact( #iqTurnTable."I/O".Outputs.Enable )
      Contact( #iqTurnTable."I/O".Outputs.Stop )
      I_Contact( #iqTurnTable."I/O".Outputs.CycleCW )
      I_Contact( #iqTurnTable."I/O".Outputs.CycleCCW )
      I_Contact( #iqTurnTable."I/O".Outputs.JogCW )
      I_Contact( #iqTurnTable."I/O".Outputs.JogCCW )
      I_Contact( #iqTurnTable."I/O".Outputs.ResetError )
      I_Contact( #iqTurnTable.Status.Collision )
      Contact( #iqTurnTable.Status.Communication )
      { S7_Templates := "SrcType := UInt" } EQ_Contact(in1 := #iqTurnTable.Status.CycleStep, in2 := 0)
      I_Contact( #iqTurnTable.Status.CycleRunning )
      I_Contact( #iqTurnTable.Status.DoneCW )
      I_Contact( #iqTurnTable.Status.DoneCCW )
      Contact( #mode_status.mode_active )
      I_Contact( #error )
      Coil( #ready_to_start )
   END_RUNG
   RUNG wire#powerrail
      Contact( #ready_to_start )
      wire#w1
      Contact( #mode_status.manual_mode )
      I_Contact( #iqTurnTable.Commands.ManualMode.JogCW )
      I_Contact( #iqTurnTable.Commands.ManualMode.JogCCW )
      wire#w2
      I_Contact( #iqTurnTable.Commands.ManualMode.StartCCW )
      Contact( #ready_to_cw )
      Coil( #iqTurnTable.Commands.ManualMode.ReadyToStartCW )
      Not()
      R_Coil( #iqTurnTable.Commands.ManualMode.StartCW )
   END_RUNG
   RUNG wire#w2
      I_Contact( #iqTurnTable.Commands.ManualMode.StartCW )
      Contact( #ready_to_ccw )
      Coil( #iqTurnTable.Commands.ManualMode.ReadyToStartCCW )
      Not()
      R_Coil( #iqTurnTable.Commands.ManualMode.StartCCW )
   END_RUNG
   RUNG wire#w1
      Contact( #mode_status.automatic_mode )
      I_Contact( #iqTurnTable.Commands.AutomaticMode.JogCW )
      I_Contact( #iqTurnTable.Commands.AutomaticMode.JogCCW )
      wire#w3
      I_Contact( #iqTurnTable.Commands.AutomaticMode.StartCCW )
      Contact( #ready_to_cw )
      Coil( #iqTurnTable.Commands.AutomaticMode.ReadyToStartCW )
      Not()
      R_Coil( #iqTurnTable.Commands.AutomaticMode.StartCW )
   END_RUNG
   RUNG wire#w3
      I_Contact( #iqTurnTable.Commands.AutomaticMode.StartCW )
      Contact( #ready_to_ccw )
      Coil( #iqTurnTable.Commands.AutomaticMode.ReadyToStartCCW )
      Not()
      R_Coil( #iqTurnTable.Commands.AutomaticMode.StartCCW )
   END_RUNG
   // the same network as SCL:
   #ready_to_start := #iPower AND #iSafety AND NOT #iReset AND NOT #iqTurnTable."I/O".Inputs.ReadyToEnable AND #iqTurnTable."I/O".Inputs.EnableActive AND #iqTurnTable."I/O".Inputs.Enabled AND #iqTurnTable."I/O".Inputs.ReadyToStart AND NOT #iqTurnTable."I/O".Inputs.Operating AND NOT #iqTurnTable."I/O".Inputs.StopIsSelected AND NOT #iqTurnTable."I/O".Inputs.STOIsSelected AND NOT #iqTurnTable."I/O".Inputs.STOIsActive AND #iqTurnTable."I/O".Outputs.Enable AND #iqTurnTable."I/O".Outputs.Stop AND NOT #iqTurnTable."I/O".Outputs.CycleCW AND NOT #iqTurnTable."I/O".Outputs.CycleCCW AND NOT #iqTurnTable."I/O".Outputs.JogCW AND NOT #iqTurnTable."I/O".Outputs.JogCCW AND NOT #iqTurnTable."I/O".Outputs.ResetError AND NOT #iqTurnTable.Status.Collision AND #iqTurnTable.Status.Communication AND (#iqTurnTable.Status.CycleStep = 0) AND NOT #iqTurnTable.Status.CycleRunning AND NOT #iqTurnTable.Status.DoneCW AND NOT #iqTurnTable.Status.DoneCCW AND #mode_status.mode_active AND NOT #error;
   #_w1 := #ready_to_start AND #mode_status.manual_mode AND NOT #iqTurnTable.Commands.ManualMode.JogCW AND NOT #iqTurnTable.Commands.ManualMode.JogCCW;
   #iqTurnTable.Commands.ManualMode.ReadyToStartCW := #_w1 AND NOT #iqTurnTable.Commands.ManualMode.StartCCW AND #ready_to_cw;
   IF NOT #iqTurnTable.Commands.ManualMode.ReadyToStartCW THEN
       #iqTurnTable.Commands.ManualMode.StartCW := FALSE;
   END_IF;
   #iqTurnTable.Commands.ManualMode.ReadyToStartCCW := #_w1 AND NOT #iqTurnTable.Commands.ManualMode.StartCW AND #ready_to_ccw;
   IF NOT #iqTurnTable.Commands.ManualMode.ReadyToStartCCW THEN
       #iqTurnTable.Commands.ManualMode.StartCCW := FALSE;
   END_IF;
   #_w2 := #ready_to_start AND #mode_status.automatic_mode AND NOT #iqTurnTable.Commands.AutomaticMode.JogCW AND NOT #iqTurnTable.Commands.AutomaticMode.JogCCW;
   #iqTurnTable.Commands.AutomaticMode.ReadyToStartCW := #_w2 AND NOT #iqTurnTable.Commands.AutomaticMode.StartCCW AND #ready_to_cw;
   IF NOT #iqTurnTable.Commands.AutomaticMode.ReadyToStartCW THEN
       #iqTurnTable.Commands.AutomaticMode.StartCW := FALSE;
   END_IF;
   #iqTurnTable.Commands.AutomaticMode.ReadyToStartCCW := #_w2 AND NOT #iqTurnTable.Commands.AutomaticMode.StartCW AND #ready_to_ccw;
   IF NOT #iqTurnTable.Commands.AutomaticMode.ReadyToStartCCW THEN
       #iqTurnTable.Commands.AutomaticMode.StartCCW := FALSE;
   END_IF;
END_REGION

REGION Network 8: Set commands
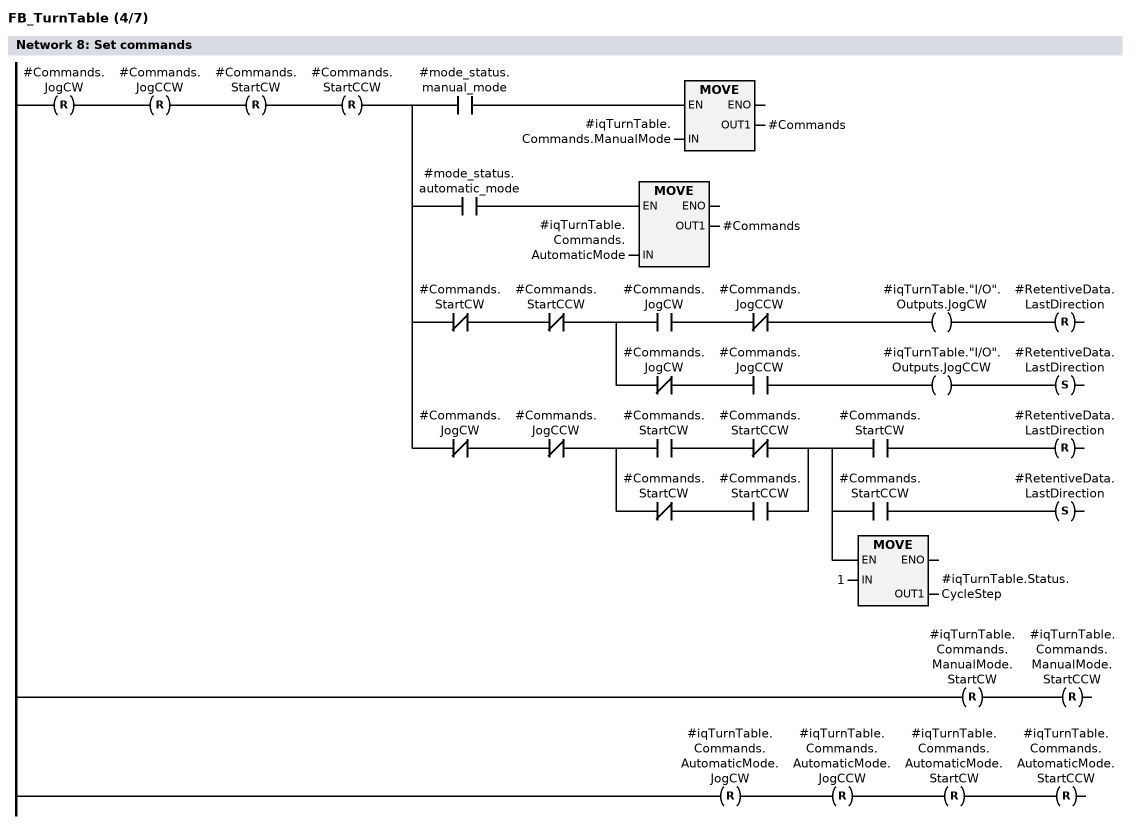
   RUNG wire#powerrail
      R_Coil( #Commands.JogCW )
      R_Coil( #Commands.JogCCW )
      R_Coil( #Commands.StartCW )
      R_Coil( #Commands.StartCCW )
      wire#w1
      Contact( #mode_status.manual_mode )
      Move(in := #iqTurnTable.Commands.ManualMode, out1 => #Commands)
   END_RUNG
   RUNG wire#w1
      Contact( #mode_status.automatic_mode )
      Move(in := #iqTurnTable.Commands.AutomaticMode, out1 => #Commands)
   END_RUNG
   RUNG wire#w1
      I_Contact( #Commands.StartCW )
      I_Contact( #Commands.StartCCW )
      wire#w2
      Contact( #Commands.JogCW )
      I_Contact( #Commands.JogCCW )
      Coil( #iqTurnTable."I/O".Outputs.JogCW )
      R_Coil( #RetentiveData.LastDirection )
   END_RUNG
   RUNG wire#w2
      I_Contact( #Commands.JogCW )
      Contact( #Commands.JogCCW )
      Coil( #iqTurnTable."I/O".Outputs.JogCCW )
      S_Coil( #RetentiveData.LastDirection )
   END_RUNG
   RUNG wire#w1
      I_Contact( #Commands.JogCW )
      I_Contact( #Commands.JogCCW )
      wire#w3
      Contact( #Commands.StartCW )
      I_Contact( #Commands.StartCCW )
      wire#w4
      Contact( #Commands.StartCW )
      R_Coil( #RetentiveData.LastDirection )
   END_RUNG
   RUNG wire#w3
      I_Contact( #Commands.StartCW )
      Contact( #Commands.StartCCW )
   END_RUNG wire#w4
   RUNG wire#w4
      Contact( #Commands.StartCCW )
      S_Coil( #RetentiveData.LastDirection )
   END_RUNG
   RUNG wire#w4
      Move(in := 1, out1 => #iqTurnTable.Status.CycleStep)
   END_RUNG
   RUNG wire#powerrail
      R_Coil( #iqTurnTable.Commands.ManualMode.StartCW )
      R_Coil( #iqTurnTable.Commands.ManualMode.StartCCW )
   END_RUNG
   RUNG wire#powerrail
      R_Coil( #iqTurnTable.Commands.AutomaticMode.JogCW )
      R_Coil( #iqTurnTable.Commands.AutomaticMode.JogCCW )
      R_Coil( #iqTurnTable.Commands.AutomaticMode.StartCW )
      R_Coil( #iqTurnTable.Commands.AutomaticMode.StartCCW )
   END_RUNG
   // the same network as SCL:
   #Commands.JogCW := FALSE;
   #Commands.JogCCW := FALSE;
   #Commands.StartCW := FALSE;
   #Commands.StartCCW := FALSE;
   IF #mode_status.manual_mode THEN #Commands := #iqTurnTable.Commands.ManualMode; END_IF;
   IF #mode_status.automatic_mode THEN #Commands := #iqTurnTable.Commands.AutomaticMode; END_IF;
   #_w1 := NOT #Commands.StartCW AND NOT #Commands.StartCCW;
   #iqTurnTable."I/O".Outputs.JogCW := #_w1 AND #Commands.JogCW AND NOT #Commands.JogCCW;
   IF #iqTurnTable."I/O".Outputs.JogCW THEN #RetentiveData.LastDirection := FALSE; END_IF;
   #iqTurnTable."I/O".Outputs.JogCCW := #_w1 AND NOT #Commands.JogCW AND #Commands.JogCCW;
   IF #iqTurnTable."I/O".Outputs.JogCCW THEN #RetentiveData.LastDirection := TRUE; END_IF;
   #_w2 := NOT #Commands.JogCW AND NOT #Commands.JogCCW AND ((#Commands.StartCW AND NOT #Commands.StartCCW) OR (NOT #Commands.StartCW AND #Commands.StartCCW));
   IF #_w2 AND #Commands.StartCW THEN #RetentiveData.LastDirection := FALSE; END_IF;
   IF #_w2 AND #Commands.StartCCW THEN #RetentiveData.LastDirection := TRUE; END_IF;
   IF #_w2 THEN #iqTurnTable.Status.CycleStep := 1; END_IF;
   #iqTurnTable.Commands.ManualMode.StartCW := FALSE;
   #iqTurnTable.Commands.ManualMode.StartCCW := FALSE;
   #iqTurnTable.Commands.AutomaticMode.JogCW := FALSE;
   #iqTurnTable.Commands.AutomaticMode.JogCCW := FALSE;
   #iqTurnTable.Commands.AutomaticMode.StartCW := FALSE;
   #iqTurnTable.Commands.AutomaticMode.StartCCW := FALSE;
END_REGION

REGION Network 9: Cycle: Reset
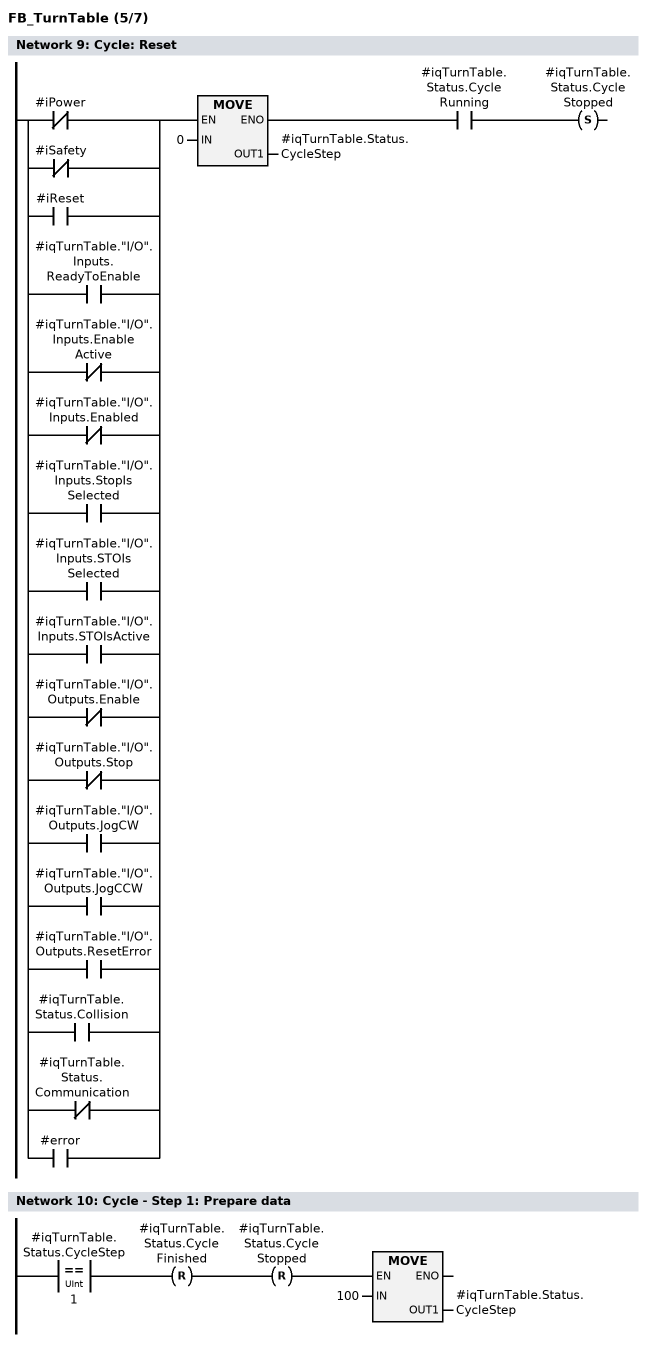
   RUNG wire#powerrail
      I_Contact( #iPower )
      wire#w1
      Move(in := 0, out1 => #iqTurnTable.Status.CycleStep)
      Contact( #iqTurnTable.Status.CycleRunning )
      S_Coil( #iqTurnTable.Status.CycleStopped )
   END_RUNG
   RUNG wire#powerrail
      I_Contact( #iSafety )
   END_RUNG wire#w1
   RUNG wire#powerrail
      Contact( #iReset )
   END_RUNG wire#w1
   RUNG wire#powerrail
      Contact( #iqTurnTable."I/O".Inputs.ReadyToEnable )
   END_RUNG wire#w1
   RUNG wire#powerrail
      I_Contact( #iqTurnTable."I/O".Inputs.EnableActive )
   END_RUNG wire#w1
   RUNG wire#powerrail
      I_Contact( #iqTurnTable."I/O".Inputs.Enabled )
   END_RUNG wire#w1
   RUNG wire#powerrail
      Contact( #iqTurnTable."I/O".Inputs.StopIsSelected )
   END_RUNG wire#w1
   RUNG wire#powerrail
      Contact( #iqTurnTable."I/O".Inputs.STOIsSelected )
   END_RUNG wire#w1
   RUNG wire#powerrail
      Contact( #iqTurnTable."I/O".Inputs.STOIsActive )
   END_RUNG wire#w1
   RUNG wire#powerrail
      I_Contact( #iqTurnTable."I/O".Outputs.Enable )
   END_RUNG wire#w1
   RUNG wire#powerrail
      I_Contact( #iqTurnTable."I/O".Outputs.Stop )
   END_RUNG wire#w1
   RUNG wire#powerrail
      Contact( #iqTurnTable."I/O".Outputs.JogCW )
   END_RUNG wire#w1
   RUNG wire#powerrail
      Contact( #iqTurnTable."I/O".Outputs.JogCCW )
   END_RUNG wire#w1
   RUNG wire#powerrail
      Contact( #iqTurnTable."I/O".Outputs.ResetError )
   END_RUNG wire#w1
   RUNG wire#powerrail
      Contact( #iqTurnTable.Status.Collision )
   END_RUNG wire#w1
   RUNG wire#powerrail
      I_Contact( #iqTurnTable.Status.Communication )
   END_RUNG wire#w1
   RUNG wire#powerrail
      Contact( #error )
   END_RUNG wire#w1
   // the same network as SCL:
   #_w1 := NOT #iPower OR NOT #iSafety OR #iReset OR #iqTurnTable."I/O".Inputs.ReadyToEnable OR NOT #iqTurnTable."I/O".Inputs.EnableActive OR NOT #iqTurnTable."I/O".Inputs.Enabled OR #iqTurnTable."I/O".Inputs.StopIsSelected OR #iqTurnTable."I/O".Inputs.STOIsSelected OR #iqTurnTable."I/O".Inputs.STOIsActive OR NOT #iqTurnTable."I/O".Outputs.Enable OR NOT #iqTurnTable."I/O".Outputs.Stop OR #iqTurnTable."I/O".Outputs.JogCW OR #iqTurnTable."I/O".Outputs.JogCCW OR #iqTurnTable."I/O".Outputs.ResetError OR #iqTurnTable.Status.Collision OR NOT #iqTurnTable.Status.Communication OR #error;
   IF #_w1 THEN #iqTurnTable.Status.CycleStep := 0; END_IF;
   IF #_w1 AND #iqTurnTable.Status.CycleRunning THEN #iqTurnTable.Status.CycleStopped := TRUE; END_IF;
END_REGION

REGION Network 10: Cycle - Step 1: Prepare data
   RUNG wire#powerrail
      { S7_Templates := "SrcType := UInt" } EQ_Contact(in1 := #iqTurnTable.Status.CycleStep, in2 := 1)
      R_Coil( #iqTurnTable.Status.CycleFinished )
      R_Coil( #iqTurnTable.Status.CycleStopped )
      Move(in := 100, out1 => #iqTurnTable.Status.CycleStep)
   END_RUNG
   // the same network as SCL:
   IF #iqTurnTable.Status.CycleStep = 1 THEN
       #iqTurnTable.Status.CycleFinished := FALSE;
       #iqTurnTable.Status.CycleStopped := FALSE;
       #iqTurnTable.Status.CycleStep := 100;
   END_IF;
END_REGION

REGION Network 11: Cycle - Step 100: Check out of position
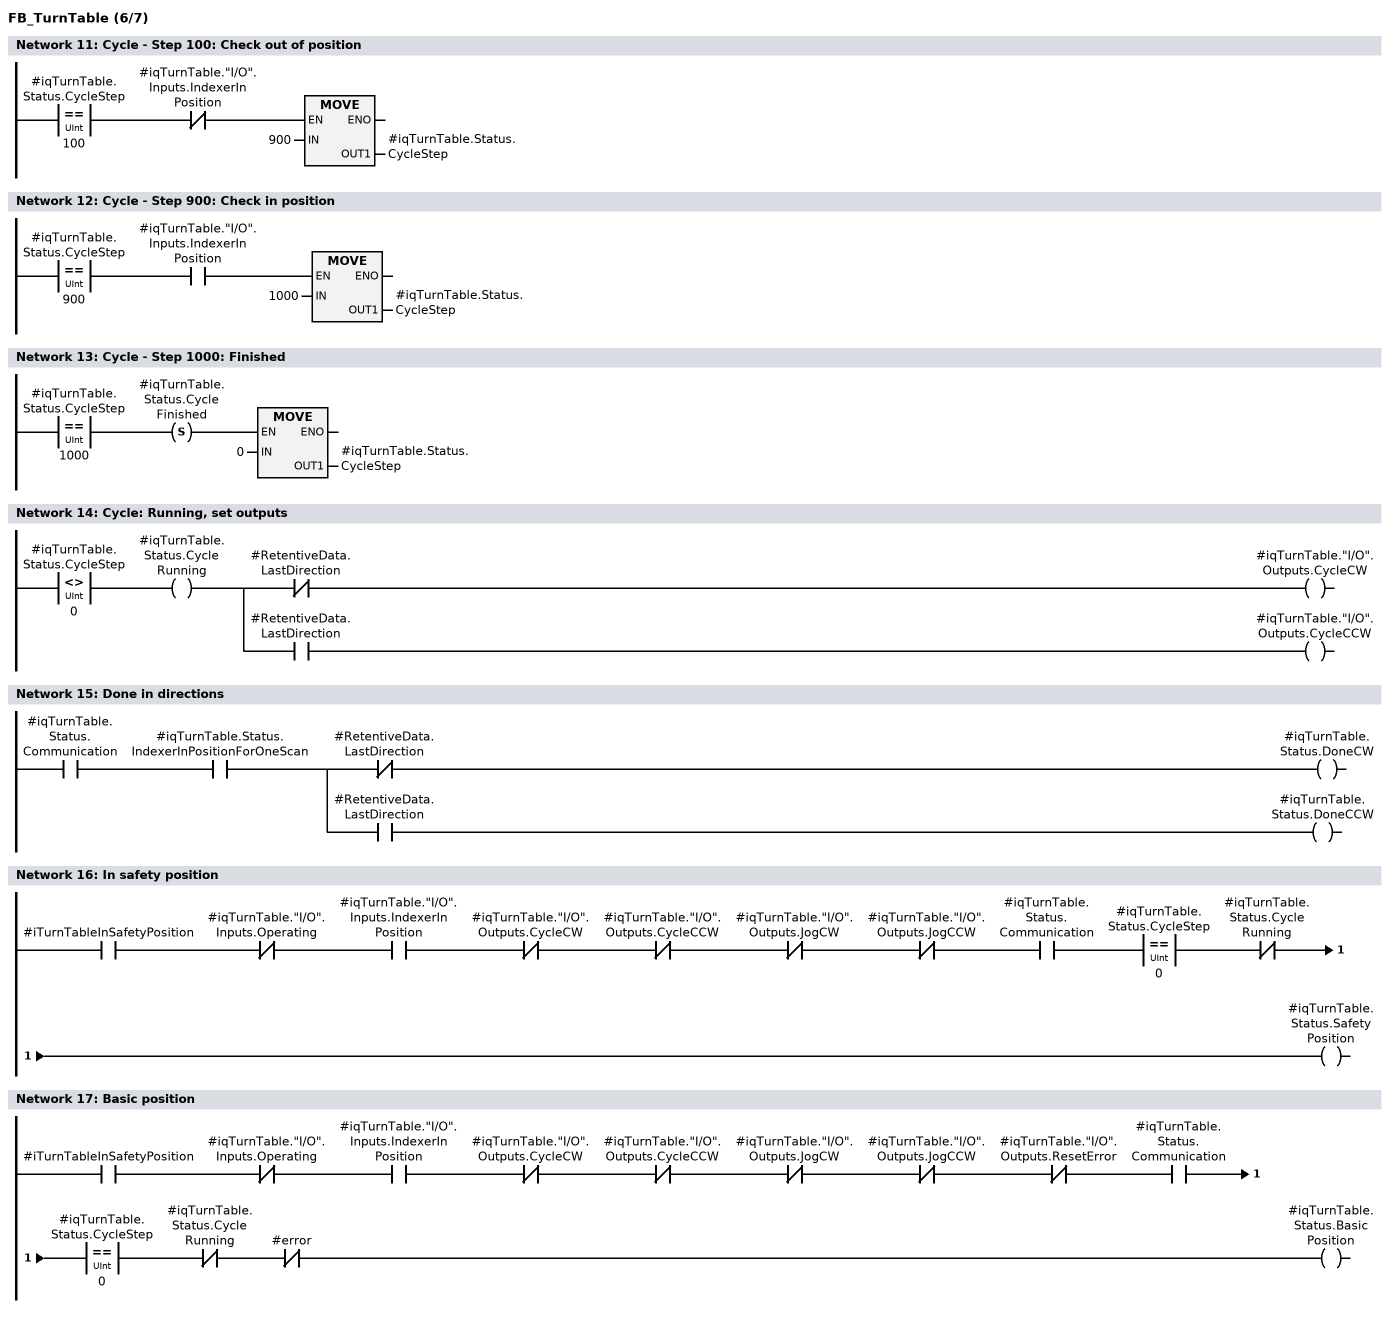
   RUNG wire#powerrail
      { S7_Templates := "SrcType := UInt" } EQ_Contact(in1 := #iqTurnTable.Status.CycleStep, in2 := 100)
      I_Contact( #iqTurnTable."I/O".Inputs.IndexerInPosition )
      Move(in := 900, out1 => #iqTurnTable.Status.CycleStep)
   END_RUNG
   // the same network as SCL:
   IF (#iqTurnTable.Status.CycleStep = 100) AND NOT #iqTurnTable."I/O".Inputs.IndexerInPosition THEN
       #iqTurnTable.Status.CycleStep := 900;
   END_IF;
END_REGION

REGION Network 12: Cycle - Step 900: Check in position
   RUNG wire#powerrail
      { S7_Templates := "SrcType := UInt" } EQ_Contact(in1 := #iqTurnTable.Status.CycleStep, in2 := 900)
      Contact( #iqTurnTable."I/O".Inputs.IndexerInPosition )
      Move(in := 1000, out1 => #iqTurnTable.Status.CycleStep)
   END_RUNG
   // the same network as SCL:
   IF (#iqTurnTable.Status.CycleStep = 900) AND #iqTurnTable."I/O".Inputs.IndexerInPosition THEN
       #iqTurnTable.Status.CycleStep := 1000;
   END_IF;
END_REGION

REGION Network 13: Cycle - Step 1000: Finished
   RUNG wire#powerrail
      { S7_Templates := "SrcType := UInt" } EQ_Contact(in1 := #iqTurnTable.Status.CycleStep, in2 := 1000)
      S_Coil( #iqTurnTable.Status.CycleFinished )
      Move(in := 0, out1 => #iqTurnTable.Status.CycleStep)
   END_RUNG
   // the same network as SCL:
   IF #iqTurnTable.Status.CycleStep = 1000 THEN
       #iqTurnTable.Status.CycleFinished := TRUE;
       #iqTurnTable.Status.CycleStep := 0;
   END_IF;
END_REGION

REGION Network 14: Cycle: Running, set outputs
   RUNG wire#powerrail
      { S7_Templates := "SrcType := UInt" } NE_Contact(in1 := #iqTurnTable.Status.CycleStep, in2 := 0)
      Coil( #iqTurnTable.Status.CycleRunning )
      wire#w1
      I_Contact( #RetentiveData.LastDirection )
      Coil( #iqTurnTable."I/O".Outputs.CycleCW )
   END_RUNG
   RUNG wire#w1
      Contact( #RetentiveData.LastDirection )
      Coil( #iqTurnTable."I/O".Outputs.CycleCCW )
   END_RUNG
   // the same network as SCL:
   #iqTurnTable.Status.CycleRunning := #iqTurnTable.Status.CycleStep <> 0;
   #iqTurnTable."I/O".Outputs.CycleCW := #iqTurnTable.Status.CycleRunning AND NOT #RetentiveData.LastDirection;
   #iqTurnTable."I/O".Outputs.CycleCCW := #iqTurnTable.Status.CycleRunning AND #RetentiveData.LastDirection;
END_REGION

REGION Network 15: Done in directions
   RUNG wire#powerrail
      Contact( #iqTurnTable.Status.Communication )
      Contact( #iqTurnTable.Status.IndexerInPositionForOneScan )
      wire#w1
      I_Contact( #RetentiveData.LastDirection )
      Coil( #iqTurnTable.Status.DoneCW )
   END_RUNG
   RUNG wire#w1
      Contact( #RetentiveData.LastDirection )
      Coil( #iqTurnTable.Status.DoneCCW )
   END_RUNG
   // the same network as SCL:
   #_w1 := #iqTurnTable.Status.Communication AND #iqTurnTable.Status.IndexerInPositionForOneScan;
   #iqTurnTable.Status.DoneCW := #_w1 AND NOT #RetentiveData.LastDirection;
   #iqTurnTable.Status.DoneCCW := #_w1 AND #RetentiveData.LastDirection;
END_REGION

REGION Network 16: In safety position
   RUNG wire#powerrail
      Contact( #iTurnTableInSafetyPosition )
      I_Contact( #iqTurnTable."I/O".Inputs.Operating )
      Contact( #iqTurnTable."I/O".Inputs.IndexerInPosition )
      I_Contact( #iqTurnTable."I/O".Outputs.CycleCW )
      I_Contact( #iqTurnTable."I/O".Outputs.CycleCCW )
      I_Contact( #iqTurnTable."I/O".Outputs.JogCW )
      I_Contact( #iqTurnTable."I/O".Outputs.JogCCW )
      Contact( #iqTurnTable.Status.Communication )
      { S7_Templates := "SrcType := UInt" } EQ_Contact(in1 := #iqTurnTable.Status.CycleStep, in2 := 0)
      I_Contact( #iqTurnTable.Status.CycleRunning )
      Coil( #iqTurnTable.Status.SafetyPosition )
   END_RUNG
   // the same network as SCL:
   #iqTurnTable.Status.SafetyPosition := #iTurnTableInSafetyPosition AND NOT #iqTurnTable."I/O".Inputs.Operating AND #iqTurnTable."I/O".Inputs.IndexerInPosition AND NOT #iqTurnTable."I/O".Outputs.CycleCW AND NOT #iqTurnTable."I/O".Outputs.CycleCCW AND NOT #iqTurnTable."I/O".Outputs.JogCW AND NOT #iqTurnTable."I/O".Outputs.JogCCW AND #iqTurnTable.Status.Communication AND (#iqTurnTable.Status.CycleStep = 0) AND NOT #iqTurnTable.Status.CycleRunning;
END_REGION

REGION Network 17: Basic position
   RUNG wire#powerrail
      Contact( #iTurnTableInSafetyPosition )
      I_Contact( #iqTurnTable."I/O".Inputs.Operating )
      Contact( #iqTurnTable."I/O".Inputs.IndexerInPosition )
      I_Contact( #iqTurnTable."I/O".Outputs.CycleCW )
      I_Contact( #iqTurnTable."I/O".Outputs.CycleCCW )
      I_Contact( #iqTurnTable."I/O".Outputs.JogCW )
      I_Contact( #iqTurnTable."I/O".Outputs.JogCCW )
      I_Contact( #iqTurnTable."I/O".Outputs.ResetError )
      Contact( #iqTurnTable.Status.Communication )
      { S7_Templates := "SrcType := UInt" } EQ_Contact(in1 := #iqTurnTable.Status.CycleStep, in2 := 0)
      I_Contact( #iqTurnTable.Status.CycleRunning )
      I_Contact( #error )
      Coil( #iqTurnTable.Status.BasicPosition )
   END_RUNG
   // the same network as SCL:
   #iqTurnTable.Status.BasicPosition := #iTurnTableInSafetyPosition AND NOT #iqTurnTable."I/O".Inputs.Operating AND #iqTurnTable."I/O".Inputs.IndexerInPosition AND NOT #iqTurnTable."I/O".Outputs.CycleCW AND NOT #iqTurnTable."I/O".Outputs.CycleCCW AND NOT #iqTurnTable."I/O".Outputs.JogCW AND NOT #iqTurnTable."I/O".Outputs.JogCCW AND NOT #iqTurnTable."I/O".Outputs.ResetError AND #iqTurnTable.Status.Communication AND (#iqTurnTable.Status.CycleStep = 0) AND NOT #iqTurnTable.Status.CycleRunning AND NOT #error;
END_REGION

REGION Network 18: Set outputs
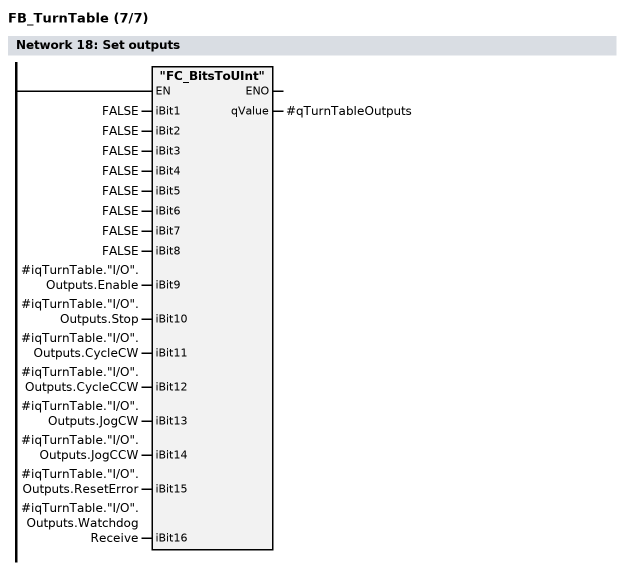
   RUNG wire#powerrail
      "FC_BitsToUInt"(iBit1 := FALSE, iBit2 := FALSE, iBit3 := FALSE, iBit4 := FALSE, iBit5 := FALSE, iBit6 := FALSE, iBit7 := FALSE, iBit8 := FALSE, iBit9 := #iqTurnTable."I/O".Outputs.Enable, iBit10 := #iqTurnTable."I/O".Outputs.Stop, iBit11 := #iqTurnTable."I/O".Outputs.CycleCW, iBit12 := #iqTurnTable."I/O".Outputs.CycleCCW, iBit13 := #iqTurnTable."I/O".Outputs.JogCW, iBit14 := #iqTurnTable."I/O".Outputs.JogCCW, iBit15 := #iqTurnTable."I/O".Outputs.ResetError, iBit16 := #iqTurnTable."I/O".Outputs.WatchdogReceive, qValue => #qTurnTableOutputs)
   END_RUNG
   // the same network as SCL:
   "FC_BitsToUInt"(iBit1 := FALSE,
                   iBit2 := FALSE,
                   iBit3 := FALSE,
                   iBit4 := FALSE,
                   iBit5 := FALSE,
                   iBit6 := FALSE,
                   iBit7 := FALSE,
                   iBit8 := FALSE,
                   iBit9 := #iqTurnTable."I/O".Outputs.Enable,
                   iBit10 := #iqTurnTable."I/O".Outputs.Stop,
                   iBit11 := #iqTurnTable."I/O".Outputs.CycleCW,
                   iBit12 := #iqTurnTable."I/O".Outputs.CycleCCW,
                   iBit13 := #iqTurnTable."I/O".Outputs.JogCW,
                   iBit14 := #iqTurnTable."I/O".Outputs.JogCCW,
                   iBit15 := #iqTurnTable."I/O".Outputs.ResetError,
                   iBit16 := #iqTurnTable."I/O".Outputs.WatchdogReceive,
                   qValue => #qTurnTableOutputs);
END_REGION
END_FUNCTION_BLOCK

FUNCTION "FC_UIntToBits" : Void   // FC1021, LAD
{ S7_Optimized_Access := 'FALSE' }
VERSION : 0.1
// stored: AutoNumber false, IsIECCheckEnabled false, SetENOAutomatically false, UDAEnableTagReadback false
   VAR_INPUT
      iValue : UInt;
   END_VAR
   VAR_OUTPUT
      qBit1 : Bool;
      qBit2 : Bool;
      qBit3 : Bool;
      qBit4 : Bool;
      qBit5 : Bool;
      qBit6 : Bool;
      qBit7 : Bool;
      qBit8 : Bool;
      qBit9 : Bool;
      qBit10 : Bool;
      qBit11 : Bool;
      qBit12 : Bool;
      qBit13 : Bool;
      qBit14 : Bool;
      qBit15 : Bool;
      qBit16 : Bool;
   END_VAR
   VAR_TEMP
      value : UInt;
   END_VAR
BEGIN

REGION Network 1: Convert UInt to bits
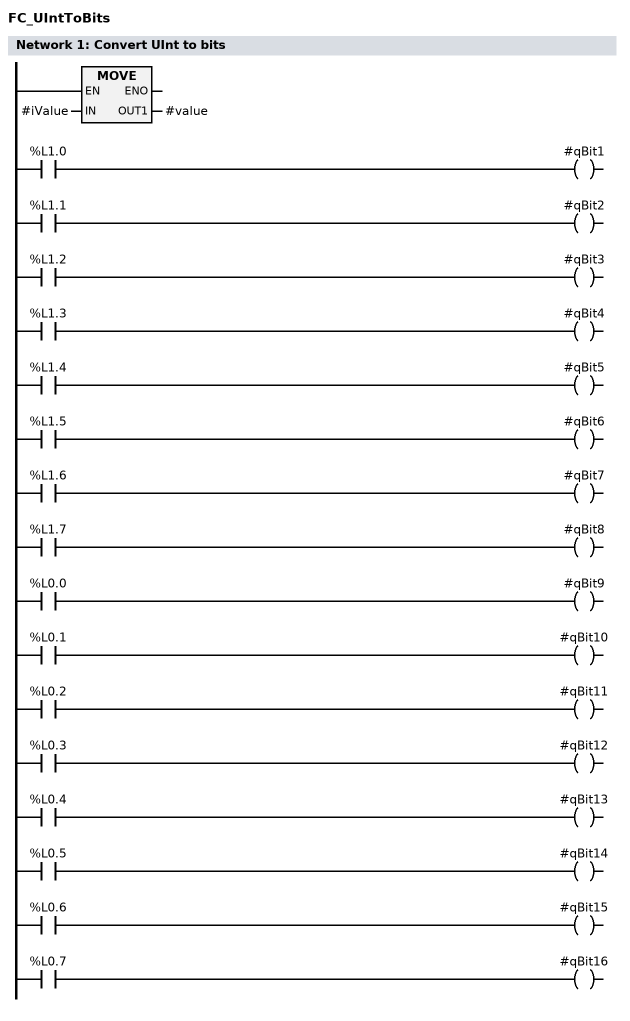
   RUNG wire#powerrail
      Move(in := #iValue, out1 => #value)
   END_RUNG
   RUNG wire#powerrail
      Contact( %L1.0 )
      Coil( #qBit1 )
   END_RUNG
   RUNG wire#powerrail
      Contact( %L1.1 )
      Coil( #qBit2 )
   END_RUNG
   RUNG wire#powerrail
      Contact( %L1.2 )
      Coil( #qBit3 )
   END_RUNG
   RUNG wire#powerrail
      Contact( %L1.3 )
      Coil( #qBit4 )
   END_RUNG
   RUNG wire#powerrail
      Contact( %L1.4 )
      Coil( #qBit5 )
   END_RUNG
   RUNG wire#powerrail
      Contact( %L1.5 )
      Coil( #qBit6 )
   END_RUNG
   RUNG wire#powerrail
      Contact( %L1.6 )
      Coil( #qBit7 )
   END_RUNG
   RUNG wire#powerrail
      Contact( %L1.7 )
      Coil( #qBit8 )
   END_RUNG
   RUNG wire#powerrail
      Contact( %L0.0 )
      Coil( #qBit9 )
   END_RUNG
   RUNG wire#powerrail
      Contact( %L0.1 )
      Coil( #qBit10 )
   END_RUNG
   RUNG wire#powerrail
      Contact( %L0.2 )
      Coil( #qBit11 )
   END_RUNG
   RUNG wire#powerrail
      Contact( %L0.3 )
      Coil( #qBit12 )
   END_RUNG
   RUNG wire#powerrail
      Contact( %L0.4 )
      Coil( #qBit13 )
   END_RUNG
   RUNG wire#powerrail
      Contact( %L0.5 )
      Coil( #qBit14 )
   END_RUNG
   RUNG wire#powerrail
      Contact( %L0.6 )
      Coil( #qBit15 )
   END_RUNG
   RUNG wire#powerrail
      Contact( %L0.7 )
      Coil( #qBit16 )
   END_RUNG
   // the same network as SCL:
   #value := #iValue;
   #qBit1 := %L1.0;
   #qBit2 := %L1.1;
   #qBit3 := %L1.2;
   #qBit4 := %L1.3;
   #qBit5 := %L1.4;
   #qBit6 := %L1.5;
   #qBit7 := %L1.6;
   #qBit8 := %L1.7;
   #qBit9 := %L0.0;
   #qBit10 := %L0.1;
   #qBit11 := %L0.2;
   #qBit12 := %L0.3;
   #qBit13 := %L0.4;
   #qBit14 := %L0.5;
   #qBit15 := %L0.6;
   #qBit16 := %L0.7;
END_REGION
END_FUNCTION

FUNCTION "FC_BitsToUInt" : Void   // FC1020, LAD
{ S7_Optimized_Access := 'FALSE' }
VERSION : 0.1
// stored: AutoNumber false, IsIECCheckEnabled false, SetENOAutomatically false, UDAEnableTagReadback false
   VAR_INPUT
      iBit1 : Bool;
      iBit2 : Bool;
      iBit3 : Bool;
      iBit4 : Bool;
      iBit5 : Bool;
      iBit6 : Bool;
      iBit7 : Bool;
      iBit8 : Bool;
      iBit9 : Bool;
      iBit10 : Bool;
      iBit11 : Bool;
      iBit12 : Bool;
      iBit13 : Bool;
      iBit14 : Bool;
      iBit15 : Bool;
      iBit16 : Bool;
   END_VAR
   VAR_OUTPUT
      qValue : UInt;
   END_VAR
   VAR_TEMP
      value : UInt;
   END_VAR
BEGIN

REGION Network 1: Convert bits to UInt
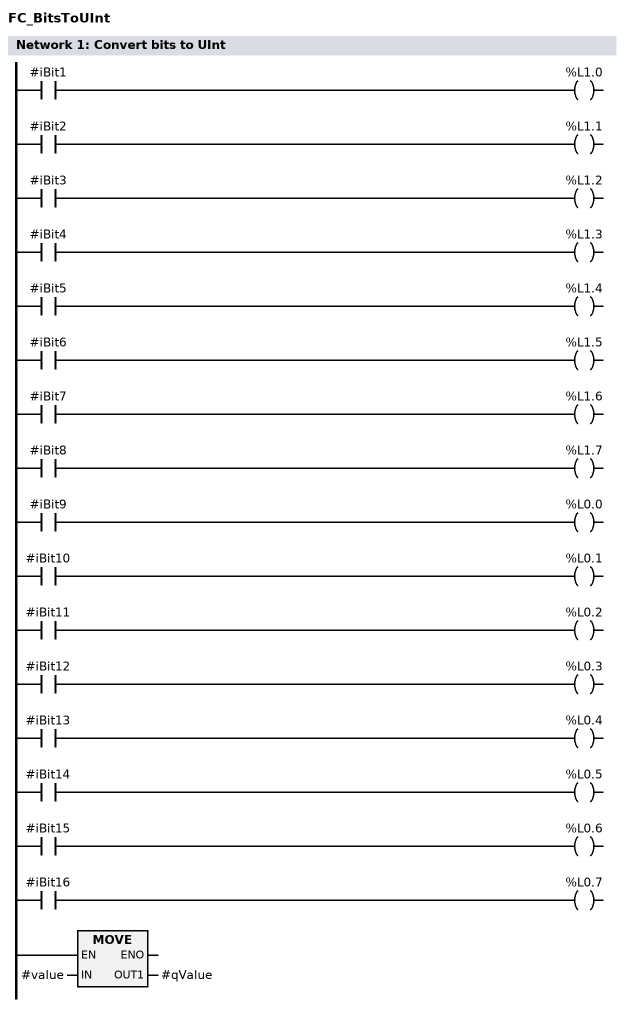
   RUNG wire#powerrail
      Contact( #iBit1 )
      Coil( %L1.0 )
   END_RUNG
   RUNG wire#powerrail
      Contact( #iBit2 )
      Coil( %L1.1 )
   END_RUNG
   RUNG wire#powerrail
      Contact( #iBit3 )
      Coil( %L1.2 )
   END_RUNG
   RUNG wire#powerrail
      Contact( #iBit4 )
      Coil( %L1.3 )
   END_RUNG
   RUNG wire#powerrail
      Contact( #iBit5 )
      Coil( %L1.4 )
   END_RUNG
   RUNG wire#powerrail
      Contact( #iBit6 )
      Coil( %L1.5 )
   END_RUNG
   RUNG wire#powerrail
      Contact( #iBit7 )
      Coil( %L1.6 )
   END_RUNG
   RUNG wire#powerrail
      Contact( #iBit8 )
      Coil( %L1.7 )
   END_RUNG
   RUNG wire#powerrail
      Contact( #iBit9 )
      Coil( %L0.0 )
   END_RUNG
   RUNG wire#powerrail
      Contact( #iBit10 )
      Coil( %L0.1 )
   END_RUNG
   RUNG wire#powerrail
      Contact( #iBit11 )
      Coil( %L0.2 )
   END_RUNG
   RUNG wire#powerrail
      Contact( #iBit12 )
      Coil( %L0.3 )
   END_RUNG
   RUNG wire#powerrail
      Contact( #iBit13 )
      Coil( %L0.4 )
   END_RUNG
   RUNG wire#powerrail
      Contact( #iBit14 )
      Coil( %L0.5 )
   END_RUNG
   RUNG wire#powerrail
      Contact( #iBit15 )
      Coil( %L0.6 )
   END_RUNG
   RUNG wire#powerrail
      Contact( #iBit16 )
      Coil( %L0.7 )
   END_RUNG
   RUNG wire#powerrail
      Move(in := #value, out1 => #qValue)
   END_RUNG
   // the same network as SCL:
   %L1.0 := #iBit1;
   %L1.1 := #iBit2;
   %L1.2 := #iBit3;
   %L1.3 := #iBit4;
   %L1.4 := #iBit5;
   %L1.5 := #iBit6;
   %L1.6 := #iBit7;
   %L1.7 := #iBit8;
   %L0.0 := #iBit9;
   %L0.1 := #iBit10;
   %L0.2 := #iBit11;
   %L0.3 := #iBit12;
   %L0.4 := #iBit13;
   %L0.5 := #iBit14;
   %L0.6 := #iBit15;
   %L0.7 := #iBit16;
   #qValue := #value;
END_REGION
END_FUNCTION

FUNCTION_BLOCK "serviceDoor"
{ S7_Optimized_Access := 'TRUE' }
VERSION : 0.1
   VAR_INPUT 
      iButtonOpen : Bool;
      iButtonLock : Bool;
      iSequenceStoped : Bool;
      iSafetyOK : Bool;
      iDoorClosed : Bool;
   END_VAR

   VAR_OUTPUT 
      qStopSequence : Bool;
      qUnlock : Bool;
      qLightOpen : Bool;
      qLightLock : Bool;
   END_VAR

   VAR 
      stopRequest : Bool;
   END_VAR


BEGIN
	IF #iSequenceStoped AND (#iButtonOpen OR #stopRequest) THEN
	    #qUnlock := TRUE;
	END_IF;
	
	IF #iButtonLock AND #iDoorClosed THEN
	    #qUnlock := FALSE;
	END_IF;
	
	IF NOT #iSequenceStoped THEN
	    IF #iButtonOpen THEN
	        #stopRequest := TRUE;
	    END_IF;
	ELSE
	    #stopRequest := FALSE;
	END_IF;
	
	#qStopSequence := #stopRequest;
	
	#qLightOpen := #qUnlock OR "Clock_1Hz" AND #stopRequest;
	#qLightLock := #iDoorClosed AND #qUnlock AND "Clock_1Hz";
	
	
	
END_FUNCTION_BLOCK

FUNCTION_BLOCK "CycleTimeMeas"   // FB46, FBD
{ S7_Optimized_Access := 'FALSE' }
VERSION : 0.1
// stored: AutoNumber false, IsIECCheckEnabled false, SetENOAutomatically false, UDAEnableTagReadback false
   VAR_INPUT
      StartCycle : Bool;
      ResetHistory : Bool;
   END_VAR
   VAR DB_SPECIFIC
      ActualTime : Time;
      LastTime : Time;
      edge2 : Bool;
      edge1 : Bool;
      Suma : DInt;
      Count : DInt;
      Max : Time;
      Min : Time;
      Average : Time;
      IEC_Timer_0_Instance { S7_SetPoint := 'True'} : TON_TIME;
      History : Array[1..20] of Time;
      NewTime : Bool;
   END_VAR
   VAR_TEMP
      d : DInt;
      i : Int;
   END_VAR
   VAR_TEMP   // added for the SCL form of the ladder/FBD networks
      _w1 : Bool;
   END_VAR
BEGIN

NETWORK
TITLE = Convert time to dint
      L     #ActualTime;
      T     #d;


REGION Network 2: Save cycle time
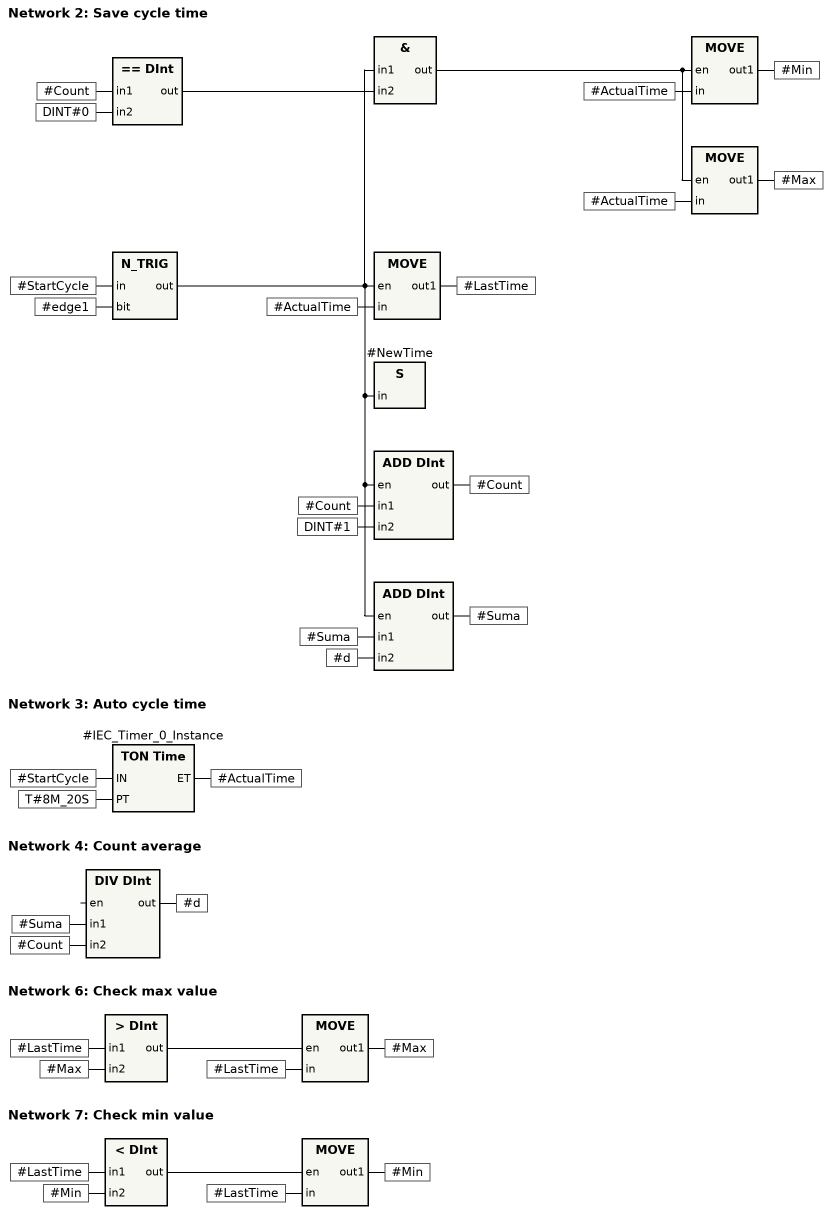
   #_w1 := NOT #StartCycle AND #edge1;   // falling edge
   #edge1 := #StartCycle;
   IF #_w1 THEN
       #LastTime := #ActualTime;
       #NewTime := TRUE;
   END_IF;
   IF #_w1 AND (#Count = DINT#0) THEN
       #Min := #ActualTime;
       #Max := #ActualTime;
   END_IF;
   IF #_w1 THEN
       #Count := #Count + DINT#1;
       #Suma := #Suma + #d;
   END_IF;
END_REGION

REGION Network 3: Auto cycle time
   #IEC_Timer_0_Instance(IN := #StartCycle, PT := T#8M_20S, ET => #ActualTime);   // TON
END_REGION

REGION Network 4: Count average
   #d := #Suma / #Count;
END_REGION

NETWORK
TITLE = Convert dint to time
      L     #d;
      T     #Average;


REGION Network 6: Check max value
   IF #LastTime > #Max THEN #Max := #LastTime; END_IF;
END_REGION

REGION Network 7: Check min value
   IF #LastTime < #Min THEN #Min := #LastTime; END_IF;
END_REGION

REGION Network 8: Reset history
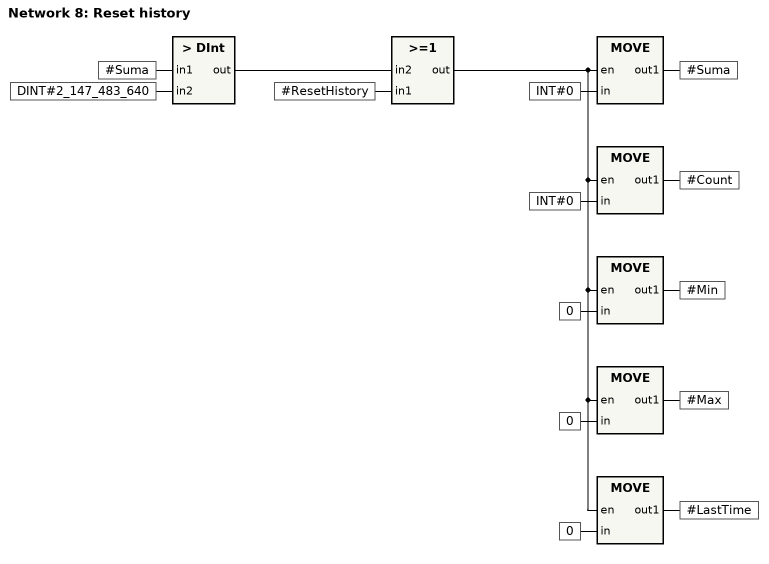
   #_w1 := (#Suma > DINT#2_147_483_640) OR #ResetHistory;
   IF #_w1 THEN
       #Suma := INT#0;
       #Count := INT#0;
       #Min := 0;
       #Max := 0;
       #LastTime := 0;
   END_IF;
END_REGION

REGION Network 10 (SCL)
   IF #NewTime THEN
       FOR #i := 1 TO 19 DO
           #History[21 - #i] := #History[20 - #i];
       END_FOR;
       #History[1] := #LastTime;
   END_IF;
   #NewTime := false;
END_REGION
END_FUNCTION_BLOCK

FUNCTION_BLOCK "FriedrichUnit"
{ S7_Optimized_Access := 'TRUE' }
VERSION : 0.1
   VAR_INPUT 
      safetyOK : Bool;
      iReady : Bool;
      iZ1OK : Bool;
      iH1OK : Bool;
      iH2OK : Bool;
      iTimeOK : Bool;
      iNoAlarm : Bool;
      FriedrichNumber : Int;
      Port : UInt;
      IP1 : USInt;
      IP2 : USInt;
      IP3 : USInt;
      IP4 : USInt;
      ID : CONN_OUC;
   END_VAR

   VAR_OUTPUT 
      qStart : Bool;
      qPrgbit4 : Bool;
      qPrgbit3 : Bool;
      qPrgbit2 : Bool;
      qPrgbit1 : Bool;
      qPrgbit0 : Bool;
      CommunicationError : Bool;
   END_VAR

   VAR_IN_OUT 
      RivetData : "UDT_Friedrich";
   END_VAR

   VAR 
      startCounter { S7_SetPoint := 'True'} : Int;
      cnt { S7_SetPoint := 'True'} : Int;
      lenghtSaved : UInt;
      R_TRIG_Start {InstructionName := 'R_TRIG'; LibVersion := '1.0'} : R_TRIG;
      IEC_Timer_Start {InstructionName := 'TON_TIME'; LibVersion := '1.0'} : TON_TIME;
      IEC_Timer_NotStarted {InstructionName := 'TON_TIME'; LibVersion := '1.0'} : TON_TIME;
      IEC_Timer_0_Error {InstructionName := 'TON_TIME'; LibVersion := '1.0'} : TON_TIME;
      ethComm : Struct
         ReconnectTimer {InstructionName := 'TON_TIME'; LibVersion := '1.0'} : TON_TIME;
         ReconnectTimer1 {InstructionName := 'TON_TIME'; LibVersion := '1.0'} : TON_TIME;
         DisableInternal { S7_SetPoint := 'True'} : Bool;
         recEnable { S7_SetPoint := 'True'} : Bool;
         recNDR : Bool;
         recBusy : Bool;
         recError : Bool;
         recStatus : Word;
         recLEN : UDInt;
         recData : Array[1..200] of Char;
         RecievedData { S7_SetPoint := 'True'} : Array[1..200] of Char;
         Connection {InstructionName := 'TCON_Param'; LibVersion := '1.0'; S7_SetPoint := 'False'} : TCON_Param;
         TS_REQ { S7_SetPoint := 'True'} : Bool;
         TS_CONT : Bool;
         TS_LEN : UDInt;
         TS_Done : Bool;
         TS_BUSY : Bool;
         TS_Error : Bool;
         TS_Status : Word;
         TS_StatusOld : Word;
         TS_Com_RST : Bool;
         DataToSend : Array[1..100] of Char;
         tConnError {InstructionName := 'TON_TIME'; LibVersion := '1.0'; S7_SetPoint := 'False'} : TON_TIME;
         s { S7_SetPoint := 'True'} : String;
         re : Real;
         d1 : DInt;
         d2 : DInt;
         lenghtSaved : UInt;
      END_STRUCT;
      TSEND_C_Instance {InstructionName := 'TSEND_C'; LibVersion := '3.2'; S7_SetPoint := 'False'} : TSEND_C;
      TRCV_Instance {InstructionName := 'TRCV'; LibVersion := '4.0'; S7_SetPoint := 'False'} : TRCV;
      IEC_Timer_start_timeout {InstructionName := 'TON_TIME'; LibVersion := '1.0'} : TON_TIME;
   END_VAR

   VAR_TEMP 
      i : Int;
      comm : Int;
      prgTemp : Int;
      s : String;
      re : Real;
   END_VAR


BEGIN
	
	(*//Start command from HMI
	IF NOT #DisableHMIControl THEN
	    #RivetData.Start := FALSE;
	    IF #HMICommand - 500 = #FriedrichNumber THEN
	        #RivetData.Start := true;
	    END_IF;
	END_IF;
	*)
	
	//Calculate program number
	IF #RivetData.PrgNumber < 1 THEN
	    #RivetData.PrgNumber := 1;
	END_IF;
	IF #RivetData.PrgNumber > 31 THEN
	    #RivetData.PrgNumber := 31;
	END_IF;
	#prgTemp := #RivetData.PrgNumber;
	#qPrgbit0 := INT_TO_BOOL(IN := #prgTemp);
	#prgTemp := SHR(IN := #prgTemp, N := 1);
	#qPrgbit1 := INT_TO_BOOL(IN := #prgTemp);
	#prgTemp := SHR(IN := #prgTemp, N := 1);
	#qPrgbit2 := INT_TO_BOOL(IN := #prgTemp);
	#prgTemp := SHR(IN := #prgTemp, N := 1);
	#qPrgbit3 := INT_TO_BOOL(IN := #prgTemp);
	#prgTemp := SHR(IN := #prgTemp, N := 1);
	#qPrgbit4 := INT_TO_BOOL(IN := #prgTemp);
	
	//Start OF riveting process
	#R_TRIG_Start(CLK := #RivetData.Start);
	IF #R_TRIG_Start.Q THEN
	    #RivetData.Start := FALSE;
	    IF #iReady THEN
	        #qStart := TRUE;
	        #RivetData.NOK := FALSE;
	        #RivetData.OK := FALSE;
	        #RivetData.Running := TRUE;
	        #RivetData.StartError := FALSE;
	        #cnt := 100;
	    END_IF;
	END_IF;
	#IEC_Timer_start_timeout(IN:=#RivetData.Start,
	                         PT:=t#1s);
	IF #IEC_Timer_start_timeout.Q THEN
	    #RivetData.Start := FALSE;
	END_IF;
	//Wait 
	#IEC_Timer_Start(IN := #cnt = 100,
	                 PT := t#500ms);
	IF #cnt = 100 THEN
	    IF #IEC_Timer_Start.Q THEN
	        #qStart := FALSE;
	        #cnt := 200;
	    END_IF;
	END_IF;
	
	//Check that riveting cycle started
	#IEC_Timer_NotStarted(IN:=#cnt=200 AND #iReady,
	                      PT:=t#1s);
	IF #cnt = 200 THEN
	    IF NOT #iReady
	    THEN
	        #cnt := 150;
	    END_IF;
	    IF #IEC_Timer_NotStarted.Q THEN
	        #qStart := TRUE;
	        #cnt := 100;
	        #startCounter := #startCounter + 1;
	        IF #startCounter > 3 THEN
	            #RivetData.StartError := TRUE;
	            #cnt := 0;
	            #RivetData.Running := FALSE;
	            #qStart := FALSE;
	        END_IF;
	    END_IF;
	END_IF;
	
	//Waiting for finished rivetin 
	IF #cnt = 150 AND #iReady THEN
	    #cnt := 160;
	END_IF;
	
	//Evaluation result
	IF #cnt = 160 THEN
	    #RivetData.Running := FALSE;
	    #RivetData.Ready := TRUE;
	    #RivetData.StartError := FALSE;
	    IF #iNoAlarm AND #iH1OK AND #iH2OK AND #iTimeOK AND #iZ1OK THEN
	        #RivetData.OK := TRUE;
	        #RivetData.NOK := FALSE;
	    ELSE
	        #RivetData.NOK := TRUE;
	        #RivetData.OK := FALSE;
	    END_IF;
	    #RivetData.H1OK := #iH1OK;
	    #RivetData.H2OK := #iH2OK;
	    #RivetData.TimeOK := #iTimeOK;
	    #RivetData.Z1OK := #iZ1OK;
	    #cnt := 0;
	END_IF;
	
	#RivetData.Ready := (#cnt = 0) AND NOT #RivetData.Start AND #iReady AND #iNoAlarm;
	
	//Alarm unit not ready   
	#IEC_Timer_0_Error(IN := (NOT #iReady OR NOT #iNoAlarm) AND #safetyOK,
	                   PT := t#15s);
	#RivetData.Error := #IEC_Timer_0_Error.Q;
	
	REGION Ethernet communication
	    REGION Connection parameters
	        #ethComm.Connection.ID := #ID;
	        #ethComm.Connection.REM_STADDR[1] := #IP1;
	        #ethComm.Connection.REM_STADDR[2] := #IP2;
	        #ethComm.Connection.REM_STADDR[3] := #IP3;
	        #ethComm.Connection.REM_STADDR[4] := #IP4;
	        
	        #ethComm.Connection.CONNECTION_TYPE := 17;
	        
	        #ethComm.d1 := UINT_TO_DINT(#Port);
	        #ethComm.d2 := #ethComm.d1 MOD 256;
	        #ethComm.d1 := #ethComm.d1 - #ethComm.d2;
	        #ethComm.d1 := #ethComm.d1 / 256;
	        
	        #ethComm.Connection.REM_TSAP_ID[1] := DINT_TO_BYTE(#ethComm.d1);
	        #ethComm.Connection.REM_TSAP_ID[2] := DINT_TO_BYTE(#ethComm.d2);
	        #ethComm.Connection.REM_STADDR_LEN := 4;
	        #ethComm.Connection.ACTIVE_EST := true;
	        #ethComm.Connection.LOCAL_DEVICE_ID := 1;
	        #ethComm.Connection.REM_TSAP_ID_LEN := 2;
	        
	        #ethComm.TS_REQ := true;
	        #ethComm.TS_CONT := NOT #ethComm.DisableInternal;
	        #ethComm.TS_LEN := 0;
	    END_REGION
	    
	    #TSEND_C_Instance(REQ := #ethComm.TS_REQ,
	                      CONT := #ethComm.TS_CONT,
	                      LEN := #ethComm.TS_LEN,
	                      DONE => #ethComm.TS_Done,
	                      BUSY => #ethComm.TS_BUSY,
	                      ERROR => #ethComm.TS_Error,
	                      STATUS => #ethComm.TS_StatusOld,
	                      CONNECT := #ethComm.Connection,
	                      DATA := #ethComm.DataToSend,
	                      COM_RST := #ethComm.TS_Com_RST);
	    
	    REGION Connection error / reconect
	        #ethComm.tConnError(IN := #ethComm.TS_StatusOld <> 16#7004,
	                            PT := t#5s,
	                            Q => #CommunicationError);
	        
	        #ethComm.ReconnectTimer(IN := #CommunicationError AND NOT #ethComm.DisableInternal,
	                                PT := t#2s);
	        IF #ethComm.ReconnectTimer.Q THEN
	            #ethComm.DisableInternal := TRUE;
	        END_IF;
	        
	        #ethComm.ReconnectTimer1(IN := #ethComm.DisableInternal,
	                                 PT := t#1s);
	        IF #ethComm.ReconnectTimer1.Q THEN
	            #ethComm.DisableInternal := FALSE;
	        END_IF;
	    END_REGION
	
	    #ethComm.recEnable := TRUE;
	    #TRCV_Instance(EN_R := #ethComm.recEnable,
	                   ID := #ID,
	                   LEN := 0,
	                   ADHOC := TRUE,
	                   NDR => #ethComm.recNDR,
	                   BUSY => #ethComm.recBusy,
	                   ERROR => #ethComm.recError,
	                   STATUS => #ethComm.recStatus,
	                   RCVD_LEN => #ethComm.recLEN,
	                   DATA := #ethComm.recData);
	    
	    REGION New data received
	        #RivetData.NewData := FALSE;
	        IF #R_TRIG_Start.Q THEN
	            #RivetData.NewDataAfterStart := FALSE;
	        END_IF;
	        IF #ethComm.recNDR THEN
	            #lenghtSaved := UDINT_TO_UINT(#ethComm.recLEN);
	            IF #lenghtSaved > 90 THEN
	                #RivetData.NewData := TRUE;
	                #RivetData.NewDataAfterStart := TRUE;
	                //Parse recieved data
	                FOR #i := 1 TO 90 DO
	                    IF #ethComm.recData[#i] = ',' THEN
	                        #ethComm.recData[#i] := '.';
	                    END_IF;
	                END_FOR;
	                
	                Chars_TO_Strg(Chars := #ethComm.recData,
	                              pChars := 18,
	                              Cnt := 5,
	                              Strg => #s);
	                #RivetData.LastTime := STRING_TO_REAL(IN := #s) * 1.0;
	                
	                Chars_TO_Strg(Chars := #ethComm.recData,
	                              pChars := 35,
	                              Cnt := 5,
	                              Strg => #s);
	                #RivetData.LastZ1 := STRING_TO_REAL(IN := #s);
	                
	                Chars_TO_Strg(Chars := #ethComm.recData,
	                              pChars := 44,
	                              Cnt := 5,
	                              Strg => #s);
	                #RivetData.LastZ2 := STRING_TO_REAL(IN := #s);
	                
	                Chars_TO_Strg(Chars := #ethComm.recData,
	                              pChars := 53,
	                              Cnt := 5,
	                              Strg => #s);
	                #RivetData.LastH1 := STRING_TO_REAL(IN := #s);
	                
	                Chars_TO_Strg(Chars := #ethComm.recData,
	                              pChars := 62,
	                              Cnt := 5,
	                              Strg => #s);
	                #RivetData.LastH2 := STRING_TO_REAL(IN := #s);
	            END_IF;
	        END_IF;
	    END_REGION
	END_REGION
	
	
END_FUNCTION_BLOCK

FUNCTION_BLOCK "RivetingCycle"   // FB52, LAD
{ S7_Optimized_Access := 'TRUE' }
VERSION : 0.1
// stored: AutoNumber true, IsIECCheckEnabled false, IsRetainMemResEnabled false, MemoryReserve 100, SetENOAutomatically false, UDAEnableTagReadback false
   VAR_INPUT
      parameters : Array[0..2] of USInt;
      basicPosition : Bool;
      twoRivets : Bool;
   END_VAR
   VAR_OUTPUT
      MeasuredData1 { ExternalAccessible := 'False'; ExternalVisible := 'False'; ExternalWritable := 'False'} : "UDT_Friedrich";
      MeasuredData2 { ExternalAccessible := 'False'; ExternalVisible := 'False'; ExternalWritable := 'False'} : "UDT_Friedrich";
   END_VAR
   VAR_IN_OUT
      riveter : "UDT_Friedrich";
      data : "UDT_FittingStatus";
      cylinderSupport : "UDT_Cylinder";
      cylinderShift : "UDT_Cylinder";
   END_VAR
   VAR
      cnt : Int;
      R_TRIG_Instance { S7_SetPoint := 'True'} : R_TRIG;
      IEC_Timer_timeout { S7_SetPoint := 'True'} : TON_TIME;
      R_TRIG_Instance_1 { S7_SetPoint := 'True'} : R_TRIG;
      ton_WayWithTimeoutReached { S7_SetPoint := 'True'} : TON_TIME;
   END_VAR
   VAR_TEMP   // added for the SCL form of the ladder/FBD networks
      _w1 : Bool;
      _w2 : Bool;
   END_VAR
BEGIN

REGION Network 1: Reset cycle
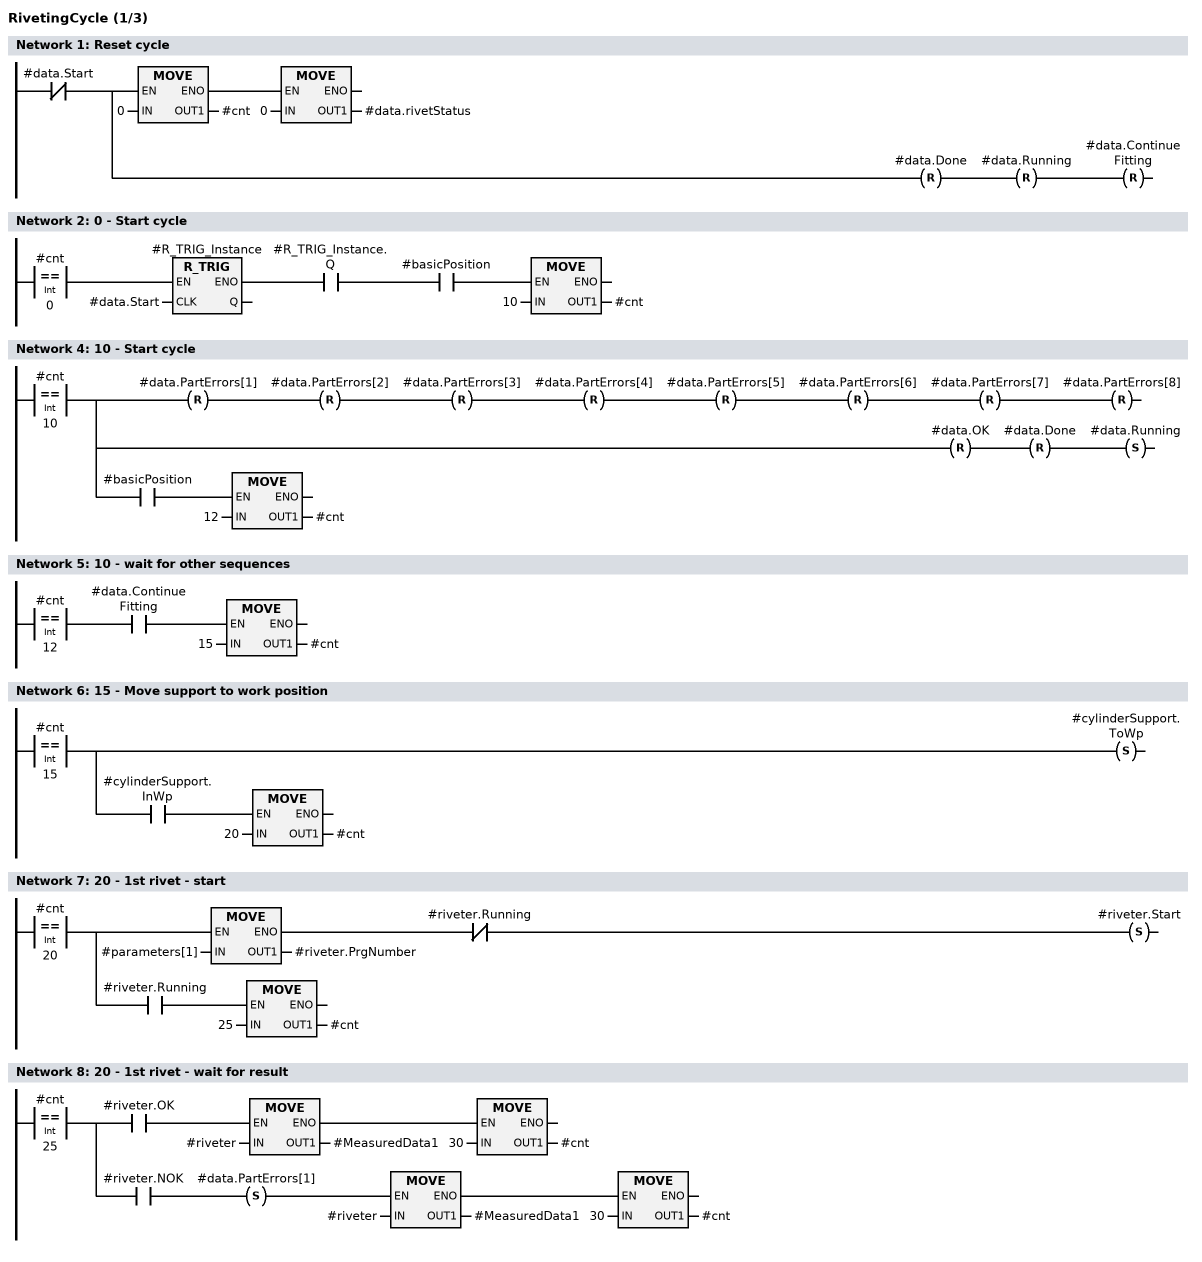
   RUNG wire#powerrail
      I_Contact( #data.Start )
      wire#w1
      Move(in := 0, out1 => #cnt)
      Move(in := 0, out1 => #data.rivetStatus)
   END_RUNG
   RUNG wire#w1
      R_Coil( #data.Done )
      R_Coil( #data.Running )
      R_Coil( #data.ContinueFitting )
   END_RUNG
   // the same network as SCL:
   IF NOT #data.Start THEN
       #cnt := 0;
       #data.rivetStatus := 0;
       #data.Done := FALSE;
       #data.Running := FALSE;
       #data.ContinueFitting := FALSE;
   END_IF;
END_REGION

REGION Network 2: 0 - Start cycle
   RUNG wire#powerrail
      { S7_Templates := "SrcType := Int" } EQ_Contact(in1 := #cnt, in2 := 0)
      #R_TRIG_Instance.R_TRIG(CLK := #data.Start, Q =>)
      Contact( #R_TRIG_Instance.Q )
      Contact( #basicPosition )
      Move(in := 10, out1 => #cnt)
   END_RUNG
   // the same network as SCL:
   #_w1 := #cnt = 0;
   #R_TRIG_Instance(EN := #_w1, CLK := #data.Start, ENO => #_w2);   // R_TRIG
   IF #_w2 AND #R_TRIG_Instance.Q AND #basicPosition THEN #cnt := 10; END_IF;
END_REGION

REGION Network 3 (SCL): 10 - Start cycle - init measured data
   IF #cnt = 10 THEN
       #MeasuredData1.Start := FALSE;
       #MeasuredData1.PrgNumber := 0;
       #MeasuredData1.Ready := FALSE;
       #MeasuredData1.Running := FALSE;
       #MeasuredData1.OK := FALSE;
       #MeasuredData1.NOK := FALSE;
       #MeasuredData1.H1OK := FALSE;
       #MeasuredData1.H2OK := FALSE;
       #MeasuredData1.TimeOK := FALSE;
       #MeasuredData1.StartError := FALSE;
       #MeasuredData1.LastH1 := 0.0;
       #MeasuredData1.LastH2 := 0.0;
       #MeasuredData1.LastTime := 0.0;
       #MeasuredData1.LastZ1 := 0.0;
       #MeasuredData1.Error := FALSE;
       #MeasuredData1.Z1OK := FALSE;
       #MeasuredData1.NewDataAfterStart := FALSE;
       #MeasuredData2 := #MeasuredData1;
   END_IF;
END_REGION

REGION Network 4: 10 - Start cycle
   RUNG wire#powerrail
      { S7_Templates := "SrcType := Int" } EQ_Contact(in1 := #cnt, in2 := 10)
      wire#w1
      R_Coil( #data.PartErrors[1] )
      R_Coil( #data.PartErrors[2] )
      R_Coil( #data.PartErrors[3] )
      R_Coil( #data.PartErrors[4] )
      R_Coil( #data.PartErrors[5] )
      R_Coil( #data.PartErrors[6] )
      R_Coil( #data.PartErrors[7] )
      R_Coil( #data.PartErrors[8] )
   END_RUNG
   RUNG wire#w1
      R_Coil( #data.OK )
      R_Coil( #data.Done )
      S_Coil( #data.Running )
   END_RUNG
   RUNG wire#w1
      Contact( #basicPosition )
      Move(in := 12, out1 => #cnt)
   END_RUNG
   // the same network as SCL:
   #_w1 := #cnt = 10;
   IF #_w1 THEN
       #data.PartErrors[1] := FALSE;
       #data.PartErrors[2] := FALSE;
       #data.PartErrors[3] := FALSE;
       #data.PartErrors[4] := FALSE;
       #data.PartErrors[5] := FALSE;
       #data.PartErrors[6] := FALSE;
       #data.PartErrors[7] := FALSE;
       #data.PartErrors[8] := FALSE;
       #data.OK := FALSE;
       #data.Done := FALSE;
       #data.Running := TRUE;
   END_IF;
   IF #_w1 AND #basicPosition THEN #cnt := 12; END_IF;
END_REGION

REGION Network 5: 10 - wait for other sequences
   RUNG wire#powerrail
      { S7_Templates := "SrcType := Int" } EQ_Contact(in1 := #cnt, in2 := 12)
      Contact( #data.ContinueFitting )
      Move(in := 15, out1 => #cnt)
   END_RUNG
   // the same network as SCL:
   IF (#cnt = 12) AND #data.ContinueFitting THEN #cnt := 15; END_IF;
END_REGION

REGION Network 6: 15 - Move support to work position
   RUNG wire#powerrail
      { S7_Templates := "SrcType := Int" } EQ_Contact(in1 := #cnt, in2 := 15)
      wire#w1
      S_Coil( #cylinderSupport.ToWp )
   END_RUNG
   RUNG wire#w1
      Contact( #cylinderSupport.InWp )
      Move(in := 20, out1 => #cnt)
   END_RUNG
   // the same network as SCL:
   #_w1 := #cnt = 15;
   IF #_w1 THEN #cylinderSupport.ToWp := TRUE; END_IF;
   IF #_w1 AND #cylinderSupport.InWp THEN #cnt := 20; END_IF;
END_REGION

REGION Network 7: 20 - 1st rivet - start
   RUNG wire#powerrail
      { S7_Templates := "SrcType := Int" } EQ_Contact(in1 := #cnt, in2 := 20)
      wire#w1
      Move(in := #parameters[1], out1 => #riveter.PrgNumber)
      I_Contact( #riveter.Running )
      S_Coil( #riveter.Start )
   END_RUNG
   RUNG wire#w1
      Contact( #riveter.Running )
      Move(in := 25, out1 => #cnt)
   END_RUNG
   // the same network as SCL:
   #_w1 := #cnt = 20;
   IF #_w1 THEN #riveter.PrgNumber := #parameters[1]; END_IF;
   IF #_w1 AND NOT #riveter.Running THEN #riveter.Start := TRUE; END_IF;
   IF #_w1 AND #riveter.Running THEN #cnt := 25; END_IF;
END_REGION

REGION Network 8: 20 - 1st rivet - wait for result
   RUNG wire#powerrail
      { S7_Templates := "SrcType := Int" } EQ_Contact(in1 := #cnt, in2 := 25)
      wire#w1
      Contact( #riveter.OK )
      Move(in := #riveter, out1 => #MeasuredData1)
      Move(in := 30, out1 => #cnt)
   END_RUNG
   RUNG wire#w1
      Contact( #riveter.NOK )
      S_Coil( #data.PartErrors[1] )
      Move(in := #riveter, out1 => #MeasuredData1)
      Move(in := 30, out1 => #cnt)
   END_RUNG
   // the same network as SCL:
   #_w1 := #cnt = 25;
   IF #_w1 AND #riveter.OK THEN
       #MeasuredData1 := #riveter;
       #cnt := 30;
   END_IF;
   IF #_w1 AND #riveter.NOK THEN
       #data.PartErrors[1] := TRUE;
       #MeasuredData1 := #riveter;
       #cnt := 30;
   END_IF;
END_REGION

REGION Network 9: 30 - Move support to base position
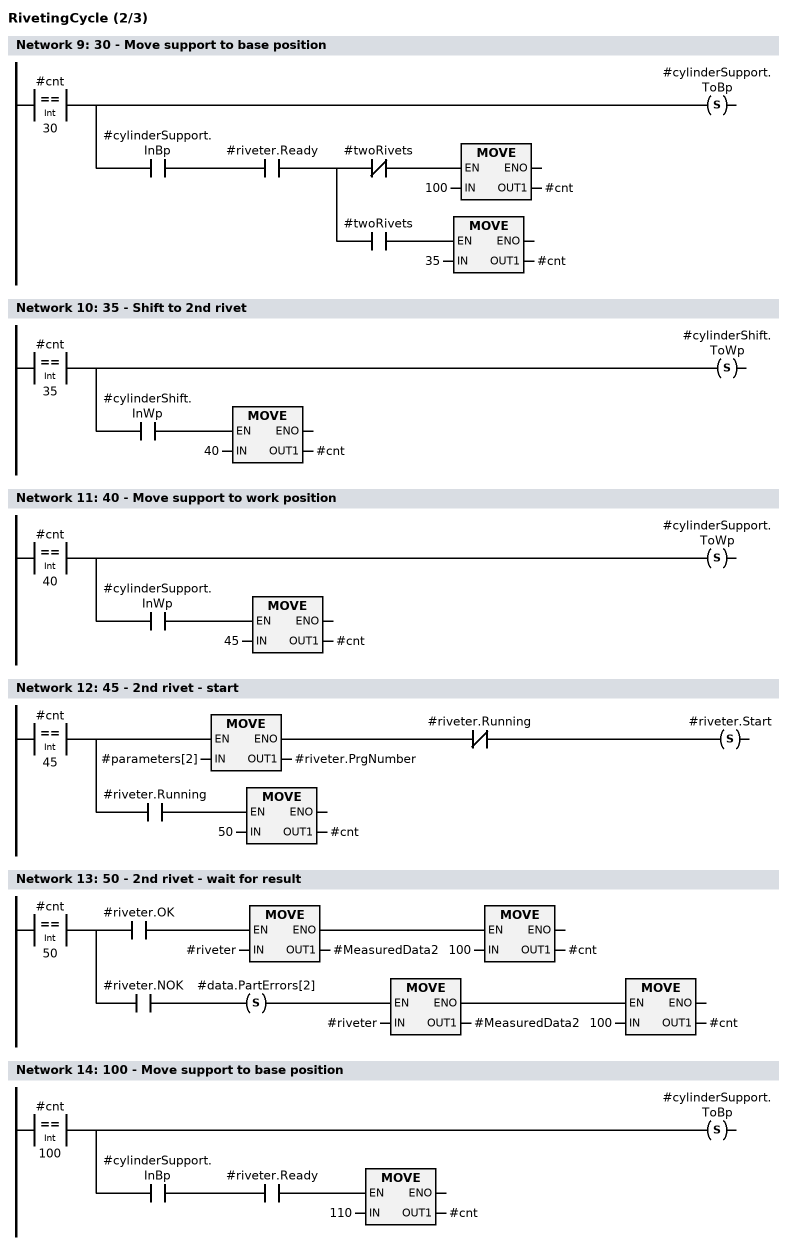
   RUNG wire#powerrail
      { S7_Templates := "SrcType := Int" } EQ_Contact(in1 := #cnt, in2 := 30)
      wire#w1
      S_Coil( #cylinderSupport.ToBp )
   END_RUNG
   RUNG wire#w1
      Contact( #cylinderSupport.InBp )
      Contact( #riveter.Ready )
      wire#w2
      I_Contact( #twoRivets )
      Move(in := 100, out1 => #cnt)
   END_RUNG
   RUNG wire#w2
      Contact( #twoRivets )
      Move(in := 35, out1 => #cnt)
   END_RUNG
   // the same network as SCL:
   #_w1 := #cnt = 30;
   IF #_w1 THEN #cylinderSupport.ToBp := TRUE; END_IF;
   #_w2 := #_w1 AND #cylinderSupport.InBp AND #riveter.Ready;
   IF #_w2 AND NOT #twoRivets THEN #cnt := 100; END_IF;
   IF #_w2 AND #twoRivets THEN #cnt := 35; END_IF;
END_REGION

REGION Network 10: 35 - Shift to 2nd rivet
   RUNG wire#powerrail
      { S7_Templates := "SrcType := Int" } EQ_Contact(in1 := #cnt, in2 := 35)
      wire#w1
      S_Coil( #cylinderShift.ToWp )
   END_RUNG
   RUNG wire#w1
      Contact( #cylinderShift.InWp )
      Move(in := 40, out1 => #cnt)
   END_RUNG
   // the same network as SCL:
   #_w1 := #cnt = 35;
   IF #_w1 THEN #cylinderShift.ToWp := TRUE; END_IF;
   IF #_w1 AND #cylinderShift.InWp THEN #cnt := 40; END_IF;
END_REGION

REGION Network 11: 40 - Move support to work position
   RUNG wire#powerrail
      { S7_Templates := "SrcType := Int" } EQ_Contact(in1 := #cnt, in2 := 40)
      wire#w1
      S_Coil( #cylinderSupport.ToWp )
   END_RUNG
   RUNG wire#w1
      Contact( #cylinderSupport.InWp )
      Move(in := 45, out1 => #cnt)
   END_RUNG
   // the same network as SCL:
   #_w1 := #cnt = 40;
   IF #_w1 THEN #cylinderSupport.ToWp := TRUE; END_IF;
   IF #_w1 AND #cylinderSupport.InWp THEN #cnt := 45; END_IF;
END_REGION

REGION Network 12: 45 - 2nd rivet - start
   RUNG wire#powerrail
      { S7_Templates := "SrcType := Int" } EQ_Contact(in1 := #cnt, in2 := 45)
      wire#w1
      Move(in := #parameters[2], out1 => #riveter.PrgNumber)
      I_Contact( #riveter.Running )
      S_Coil( #riveter.Start )
   END_RUNG
   RUNG wire#w1
      Contact( #riveter.Running )
      Move(in := 50, out1 => #cnt)
   END_RUNG
   // the same network as SCL:
   #_w1 := #cnt = 45;
   IF #_w1 THEN #riveter.PrgNumber := #parameters[2]; END_IF;
   IF #_w1 AND NOT #riveter.Running THEN #riveter.Start := TRUE; END_IF;
   IF #_w1 AND #riveter.Running THEN #cnt := 50; END_IF;
END_REGION

REGION Network 13: 50 - 2nd rivet - wait for result
   RUNG wire#powerrail
      { S7_Templates := "SrcType := Int" } EQ_Contact(in1 := #cnt, in2 := 50)
      wire#w1
      Contact( #riveter.OK )
      Move(in := #riveter, out1 => #MeasuredData2)
      Move(in := 100, out1 => #cnt)
   END_RUNG
   RUNG wire#w1
      Contact( #riveter.NOK )
      S_Coil( #data.PartErrors[2] )
      Move(in := #riveter, out1 => #MeasuredData2)
      Move(in := 100, out1 => #cnt)
   END_RUNG
   // the same network as SCL:
   #_w1 := #cnt = 50;
   IF #_w1 AND #riveter.OK THEN
       #MeasuredData2 := #riveter;
       #cnt := 100;
   END_IF;
   IF #_w1 AND #riveter.NOK THEN
       #data.PartErrors[2] := TRUE;
       #MeasuredData2 := #riveter;
       #cnt := 100;
   END_IF;
END_REGION

REGION Network 14: 100 - Move support to base position
   RUNG wire#powerrail
      { S7_Templates := "SrcType := Int" } EQ_Contact(in1 := #cnt, in2 := 100)
      wire#w1
      S_Coil( #cylinderSupport.ToBp )
   END_RUNG
   RUNG wire#w1
      Contact( #cylinderSupport.InBp )
      Contact( #riveter.Ready )
      Move(in := 110, out1 => #cnt)
   END_RUNG
   // the same network as SCL:
   #_w1 := #cnt = 100;
   IF #_w1 THEN #cylinderSupport.ToBp := TRUE; END_IF;
   IF #_w1 AND #cylinderSupport.InBp AND #riveter.Ready THEN #cnt := 110; END_IF;
END_REGION

REGION Network 15: 110 - Shift to base position
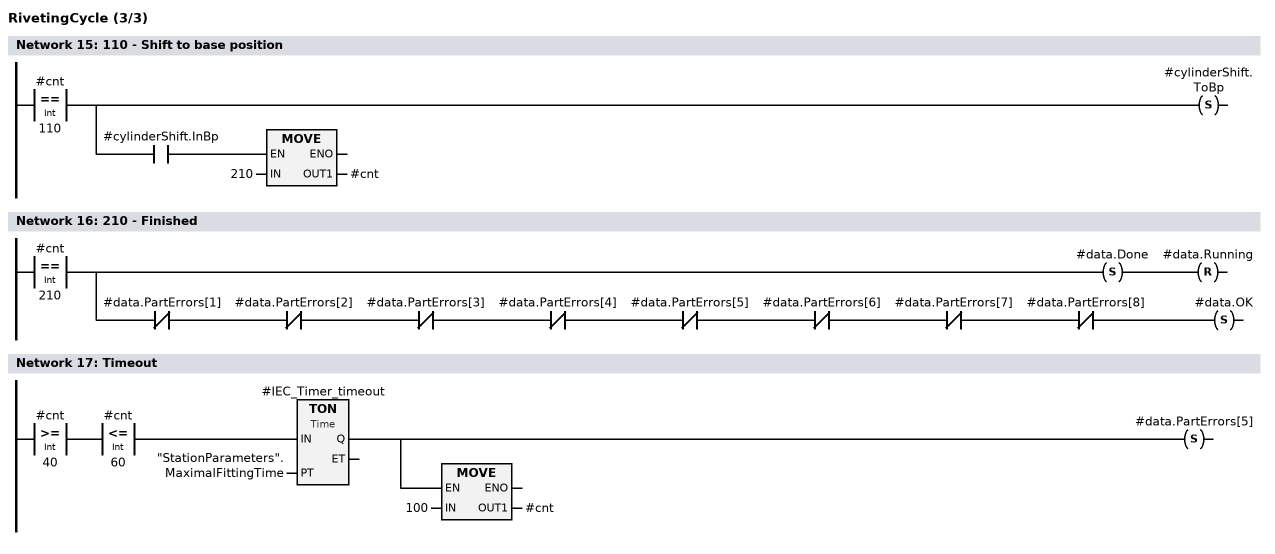
   RUNG wire#powerrail
      { S7_Templates := "SrcType := Int" } EQ_Contact(in1 := #cnt, in2 := 110)
      wire#w1
      S_Coil( #cylinderShift.ToBp )
   END_RUNG
   RUNG wire#w1
      Contact( #cylinderShift.InBp )
      Move(in := 210, out1 => #cnt)
   END_RUNG
   // the same network as SCL:
   #_w1 := #cnt = 110;
   IF #_w1 THEN #cylinderShift.ToBp := TRUE; END_IF;
   IF #_w1 AND #cylinderShift.InBp THEN #cnt := 210; END_IF;
END_REGION

REGION Network 16: 210 - Finished
   RUNG wire#powerrail
      { S7_Templates := "SrcType := Int" } EQ_Contact(in1 := #cnt, in2 := 210)
      wire#w1
      S_Coil( #data.Done )
      R_Coil( #data.Running )
   END_RUNG
   RUNG wire#w1
      I_Contact( #data.PartErrors[1] )
      I_Contact( #data.PartErrors[2] )
      I_Contact( #data.PartErrors[3] )
      I_Contact( #data.PartErrors[4] )
      I_Contact( #data.PartErrors[5] )
      I_Contact( #data.PartErrors[6] )
      I_Contact( #data.PartErrors[7] )
      I_Contact( #data.PartErrors[8] )
      S_Coil( #data.OK )
   END_RUNG
   // the same network as SCL:
   #_w1 := #cnt = 210;
   IF #_w1 THEN
       #data.Done := TRUE;
       #data.Running := FALSE;
   END_IF;
   IF #_w1 AND NOT #data.PartErrors[1] AND NOT #data.PartErrors[2] AND NOT #data.PartErrors[3] AND NOT #data.PartErrors[4] AND NOT #data.PartErrors[5] AND NOT #data.PartErrors[6] AND NOT #data.PartErrors[7] AND NOT #data.PartErrors[8] THEN
       #data.OK := TRUE;
   END_IF;
END_REGION

REGION Network 17: Timeout
   RUNG wire#powerrail
      { S7_Templates := "SrcType := Int" } GE_Contact(in1 := #cnt, in2 := 40)
      { S7_Templates := "SrcType := Int" } LE_Contact(in1 := #cnt, in2 := 60)
      { S7_Templates := "time_type := Time" } #IEC_Timer_timeout.TON(pt := "StationParameters".MaximalFittingTime, et =>)
      wire#w1
      S_Coil( #data.PartErrors[5] )
   END_RUNG
   RUNG wire#w1
      Move(in := 100, out1 => #cnt)
   END_RUNG
   // the same network as SCL:
   #IEC_Timer_timeout(IN := (#cnt >= 40) AND (#cnt <= 60), PT := "StationParameters".MaximalFittingTime);   // TON
   IF #IEC_Timer_timeout.Q THEN
       #data.PartErrors[5] := TRUE;
       #cnt := 100;
   END_IF;
END_REGION
END_FUNCTION_BLOCK

FUNCTION_BLOCK "Camera"
{ S7_Optimized_Access := 'TRUE' }
VERSION : 0.1
   VAR_INPUT 
      Command_Control_Address : HW_IO;
      Command_Status_Bits_Address : HW_IO;
      Device_Result_Bits_Address : HW_IO;
      Device_Status_Words_Address : HW_IO;
      Device_Statistics_Address : HW_IO;
      Position_Adjust_Result_Address : HW_IO;
   END_VAR

   VAR_IN_OUT 
      data : "UDT_Camera_Keyence_IV";
   END_VAR

   VAR 
      state : Int;
      OKCount : Int;
      NOKCount : Int;
      Command_Control : Struct
         Trigger_request : Bool;
         Master_registration_request : Bool;
         Program_switching_request : Bool;
         Warning_clear_request : Bool;
         Statistics_reset_request : Bool;
         Buffer_clear_request : Bool;
         reserve1 : Bool;
         reserve2 : Bool;
         reserve3 : Bool;
         reserve4 : Bool;
         reserve5 : Bool;
         reserve6 : Bool;
         reserve7 : Bool;
         reserve8 : Bool;
         reserve9 : Bool;
         reserve10 : Bool;
         Result_acquisition_complete_notification : Bool;
         reserve11 : Bool;
         reserve12 : Bool;
         reserve13 : Bool;
         reserve14 : Bool;
         reserve15 : Bool;
         reserve16 : Bool;
         reserve17 : Bool;
         reserve18 : Bool;
         reserve19 : Bool;
         reserve20 : Bool;
         reserve21 : Bool;
         reserve22 : Bool;
         reserve23 : Bool;
         reserve24 : Bool;
         reserve25 : Bool;
         ProgramNumber : UInt;
         reserve : Array[1..6] of Byte;
      END_STRUCT;
      Command_Status_Bits : Struct
         Trigger_response : Bool;
         Master_registration_response : Bool;
         Program_switching_response : Bool;
         Warning_clear_response : Bool;
         Statistics_reset_response : Bool;
         Buffer_clear_response : Bool;
         reserve1 : Bool;
         reserve2 : Bool;
         Trigger_failed : Bool;
         Master_registration_failed : Bool;
         Program_switching_failed : Bool;
         reserve3 : Bool;
         reserve4 : Bool;
         reserve5 : Bool;
         reserve6 : Bool;
         reserve7 : Bool;
         Result_available : Bool;
         Result_update_complete : Bool;
         BUSY : Bool;
         Imaging_status : Bool;
         RUN : Bool;
         Ready : Bool;
         reserve8 : Bool;
         reserve9 : Bool;
         reserve10 : Bool;
         reserve11 : Bool;
         reserve12 : Bool;
         reserve13 : Bool;
         reserve14 : Bool;
         Buffer_overrun : Bool;
         Warning : Bool;
         Error : Bool;
      END_STRUCT;
      Device_Result_Bits : Struct
         Overall_judgment : Bool;
         Position_correction : Bool;
         LOGIC1 : Bool;
         LOGIC2 : Bool;
         LOGIC3 : Bool;
         LOGIC4 : Bool;
         Overall_judgment_NG : Bool;
         reserve1 : Bool;
         reserve2 : Bool;
         reserve3 : Bool;
         reserve4 : Bool;
         reserve5 : Bool;
         reserve6 : Bool;
         reserve7 : Bool;
         reserve8 : Bool;
         Tool : Array[1..16] of Bool;
      END_STRUCT;
      Device_Status_Words : Struct
         Error_No : UInt;
         Warning_No : UInt;
         Nimber_of_remaining_buffers : UInt;
         Checksum : UInt;
         Current_program : UInt;
         Program_No_during_judgment : UInt;
         Result_No : UInt;
         Processing_time : UInt;
      END_STRUCT;
      IEC_Timer_0_zmenaProgramu {InstructionName := 'TON_TIME'; LibVersion := '1.0'} : TON_TIME;
      IEC_Timer_0_Instance {InstructionName := 'TON_TIME'; LibVersion := '1.0'} : TON_TIME;
      ton_NextTry {InstructionName := 'TON_TIME'; LibVersion := '1.0'} : TON_TIME;
      Result_update_complete_mem { S7_SetPoint := 'True'} : Bool;
      Trigger_request_mem : Bool;
      R_TRIG_Instance {InstructionName := 'R_TRIG'; LibVersion := '1.0'} : R_TRIG;
      IEC_Timer_Results_timeout {InstructionName := 'TON_TIME'; LibVersion := '1.0'} : TON_TIME;
   END_VAR

   VAR_TEMP 
      retValTmp : Int;
      i : Int;
   END_VAR


BEGIN
	#retValTmp := DPRD_DAT(LADDR := #Command_Status_Bits_Address, RECORD => #Command_Status_Bits);
	#retValTmp := DPRD_DAT(LADDR := #Device_Result_Bits_Address, RECORD => #Device_Result_Bits);
	#retValTmp := DPRD_DAT(LADDR := #Device_Status_Words_Address, RECORD => #Device_Status_Words);
	
	#Command_Control.ProgramNumber := SINT_TO_UINT(#data.ProgramNumber);
	#data.ProgramOK := #Command_Control.ProgramNumber = #Device_Status_Words.Current_program;
	#Command_Control.Program_switching_request := NOT #data.ProgramOK AND "Clock_10Hz";
	#IEC_Timer_0_zmenaProgramu(IN := NOT #data.ProgramOK,
	                           PT := t#10s,
	                           Q => #data.ProgramChangeNOK);
	
	#Command_Control.Trigger_request := #data.Start AND #data.ProgramOK AND "Clock_10Hz";
	#R_TRIG_Instance(CLK:=#Command_Control.Trigger_request);
	IF #R_TRIG_Instance.Q (*OR NOT #data.Start*) THEN
	    #data.Result := 0;
	END_IF;
	
	REGION #init tool results
	    IF NOT #data.ProgramOK THEN
	        FOR #i := 1 TO 16 DO
	            #data.Tool[#i] := FALSE;
	        END_FOR;
	        #data.Result := 0;
	        #data.ResultReadyAfterChange := FALSE;
	    END_IF;
	END_REGION
	
	#IEC_Timer_Results_timeout(IN := #Command_Status_Bits.Result_update_complete = #Result_update_complete_mem,
	                           PT := t#300ms);
	IF #IEC_Timer_Results_timeout.Q THEN
	    #data.Result := 0;
	END_IF;
	
	REGION read tool results
	    IF #Command_Status_Bits.Result_update_complete <> #Result_update_complete_mem AND #data.ProgramOK THEN
	        #data.Tool := #Device_Result_Bits.Tool;
	        IF #Device_Result_Bits.Overall_judgment THEN
	            #data.Result := 1;
	        ELSE
	            #data.Result := -1;
	        END_IF;
	        #data.ResultReadyAfterChange := TRUE;
	    END_IF;
	END_REGION
	
	    
	#Result_update_complete_mem := #Command_Status_Bits.Result_update_complete;
	#Trigger_request_mem := #Command_Control.Trigger_request;
	
	#retValTmp := DPWR_DAT(LADDR := #Command_Control_Address, RECORD := #Command_Control);
	
END_FUNCTION_BLOCK

FUNCTION_BLOCK "SlidesMain"   // FB25, LAD
{ S7_Optimized_Access := 'TRUE' }
VERSION : 0.1
// stored: AutoNumber true, IsIECCheckEnabled false, IsRetainMemResEnabled false, MemoryReserve 100, SetENOAutomatically false, UDAEnableTagReadback false
   VAR
      R_TRIG_Instance { S7_SetPoint := 'True'} : R_TRIG;
      IEC_Timer_0_Instance { S7_SetPoint := 'True'} : TON_TIME;
      IEC_Timer_0_Instance_1 { S7_SetPoint := 'True'} : TOF_TIME;
      IEC_Timer_0_Instance_3 { S7_SetPoint := 'True'} : TON_TIME;
      IEC_Timer_0_Instance_5 { S7_SetPoint := 'True'} : TON_TIME;
   END_VAR
BEGIN

REGION Network 1 (SCL): NOK box from part holders
   //Check amount of parts in stock
   IF "PartHolderData".NOKBoxAmount >= "StationParameters".NOKBoxSize THEN
       "PartHolderData".NOKBoxFull := true;
   ELSE
       "PartHolderData".NOKBoxFull := FALSE;
   END_IF;

   //NOK Box signal with delay
   #R_TRIG_Instance(CLK:=NOT "iNokPartOpticalSensor");
   IF #R_TRIG_Instance.Q THEN
       "PartHolderData".NOKBoxActivated := true;
   END_IF;
   #IEC_Timer_0_Instance(IN:="PartHolderData".NOKBoxActivated,
                         PT:=t#2s);
   IF #IEC_Timer_0_Instance.Q THEN
       "PartHolderData".NOKBoxActivated := false;
   END_IF;

   //Box presence with delay
   #IEC_Timer_0_Instance_1(IN:="iNokBoxPresent",
                           PT:=t#1s,
                           Q=>"PartHolderData".NOKBoxPesent);

   //Error NOK box signal sensor
   #IEC_Timer_0_Instance_3(IN:=NOT "iNokPartOpticalSensor",
                           PT:=t#3s);
   IF #IEC_Timer_0_Instance_3.Q AND "PartHolderData".NOKBoxPesent THEN
       "SetAlarm"(AlarmNumber := 42,
                  Cell := 1,
                  Station := 99);
       ;
   END_IF;

   #IEC_Timer_0_Instance_5(IN:=NOT "iNokBoxPresent",
                           PT:=t#3s);
   IF #IEC_Timer_0_Instance_5.Q THEN
       "SetAlarm"(AlarmNumber := 40,
                  Cell := 1,
                  Station := 99);
       ;
   END_IF;

   IF "PartHolderData".NOKBoxFull THEN
       "SetAlarm"(AlarmNumber := 43,
                  Cell := 1,
                  Station := 99);
   END_IF;

   //Reset holders amounts
   "PartHolderData".ConfirmEmptyNOKBox := "PartHolderData".NOKBoxFull;
   IF "PartHolderData".EmptyNOKBoxConfirmed THEN
       "PartHolderData".NOKBoxAmount := 0;
   END_IF;
   "PartHolderData".EmptyNOKBoxConfirmed := false;
END_REGION
END_FUNCTION_BLOCK

FUNCTION_BLOCK "ModeSelection"   // FB38, GRAPH
VERSION : 0.1
// stored: AcknowledgeErrorsRequired true, AutoNumber true, GraphVersion 6.0, InitialValuesAcquisition false, IsIECCheckEnabled false, LanguageInNetworks LAD, LockOperatingMode false, PermanentILProcessingInMANMode false, SetENOAutomatically false, SkipSteps false, UDAEnableTagReadback false, WithAlarmHandling true
   // inherited from GRAPH_BASE
   VAR
      OFF_SQ_BASE : Bool;
   END_VAR
   VAR_INPUT
      iSafetyOKauto : Bool;
      iSafetyOKmanual : Bool;
      iBasePosition : Bool;
      iPozadavekZastavitOdDveri : Bool;
      iLinkaZastavena : Bool;
      iLinkaPrazdna : Bool;
      iBaseInManualMode : Bool;
      OFF_SQ { ExternalAccessible := 'False'; ExternalVisible := 'False'; ExternalWritable := 'False'} : Bool := false;   // Turn sequence off
      INIT_SQ { ExternalAccessible := 'False'; ExternalVisible := 'False'; ExternalWritable := 'False'} : Bool := false;   // Set sequence to initial state
      ACK_EF { ExternalAccessible := 'False'; ExternalVisible := 'False'; ExternalWritable := 'False'} : Bool := false;   // Acknowledge all errors and faults
      S_PREV { ExternalAccessible := 'False'; ExternalVisible := 'False'; ExternalWritable := 'False'} : Bool := false;   // Output previous step in parameter S_NO
      S_NEXT { ExternalAccessible := 'False'; ExternalVisible := 'False'; ExternalWritable := 'False'} : Bool := false;   // Indicate next step in parameter S_NO
      SW_AUTO { ExternalAccessible := 'False'; ExternalVisible := 'False'; ExternalWritable := 'False'} : Bool := false;   // Automatic mode
      SW_TAP { ExternalAccessible := 'False'; ExternalVisible := 'False'; ExternalWritable := 'False'} : Bool := false;   // Semiautomatic/switch with transition
      SW_TOP { ExternalAccessible := 'False'; ExternalVisible := 'False'; ExternalWritable := 'False'} : Bool := false;   // Semiautomatic/ignore transition
      SW_MAN { ExternalAccessible := 'False'; ExternalVisible := 'False'; ExternalWritable := 'False'} : Bool := false;   // Manual mode
      S_SEL { ExternalAccessible := 'False'; ExternalVisible := 'False'; ExternalWritable := 'False'} : Int := 0;   // Select step to be output to S_NO
      S_ON { ExternalAccessible := 'False'; ExternalVisible := 'False'; ExternalWritable := 'False'} : Bool := false;   // Activate step indicated in S_NO
      S_OFF { ExternalAccessible := 'False'; ExternalVisible := 'False'; ExternalWritable := 'False'} : Bool := false;   // Deactivate step indicated S_NO
      T_PUSH { ExternalAccessible := 'False'; ExternalVisible := 'False'; ExternalWritable := 'False'} : Bool := false;   // Enable transition to switch in semi automatic mode
   END_VAR
   VAR_OUTPUT
      S_NO { ExternalAccessible := 'False'; ExternalVisible := 'False'; ExternalWritable := 'False'} : Int := 0;   // Step number
      S_MORE { ExternalAccessible := 'False'; ExternalVisible := 'False'; ExternalWritable := 'False'} : Bool := false;   // More steps are available and can be shown in S_NO
      S_ACTIVE { ExternalAccessible := 'False'; ExternalVisible := 'False'; ExternalWritable := 'False'} : Bool := false;   // Step indicated in S_NO is active
      ERR_FLT { ExternalAccessible := 'False'; ExternalVisible := 'False'; ExternalWritable := 'False'} : Bool := false;   // Interlock or supervision group error
      AUTO_ON { ExternalAccessible := 'False'; ExternalVisible := 'False'; ExternalWritable := 'False'} : Bool := false;   // Automatic mode is active
      TAP_ON { ExternalAccessible := 'False'; ExternalVisible := 'False'; ExternalWritable := 'False'} : Bool := false;   // Semiautomatic mode/step with transition enabled
      TOP_ON { ExternalAccessible := 'False'; ExternalVisible := 'False'; ExternalWritable := 'False'} : Bool := false;   // Semiautomatic mode/ignore transition enabled
      MAN_ON { ExternalAccessible := 'False'; ExternalVisible := 'False'; ExternalWritable := 'False'} : Bool := false;   // Manual mode is active
   END_VAR
   VAR
      dummy : Bool;
   END_VAR
   VAR RETAIN
      mode : "udtModes";
   END_VAR
   VAR
      PrevMode : Int;
      F_TRIG_semiauto_switch { S7_SetPoint := 'True'} : F_TRIG;
      F_TRIG_switchAuto { S7_SetPoint := 'True'} : F_TRIG;
   END_VAR
BEGIN
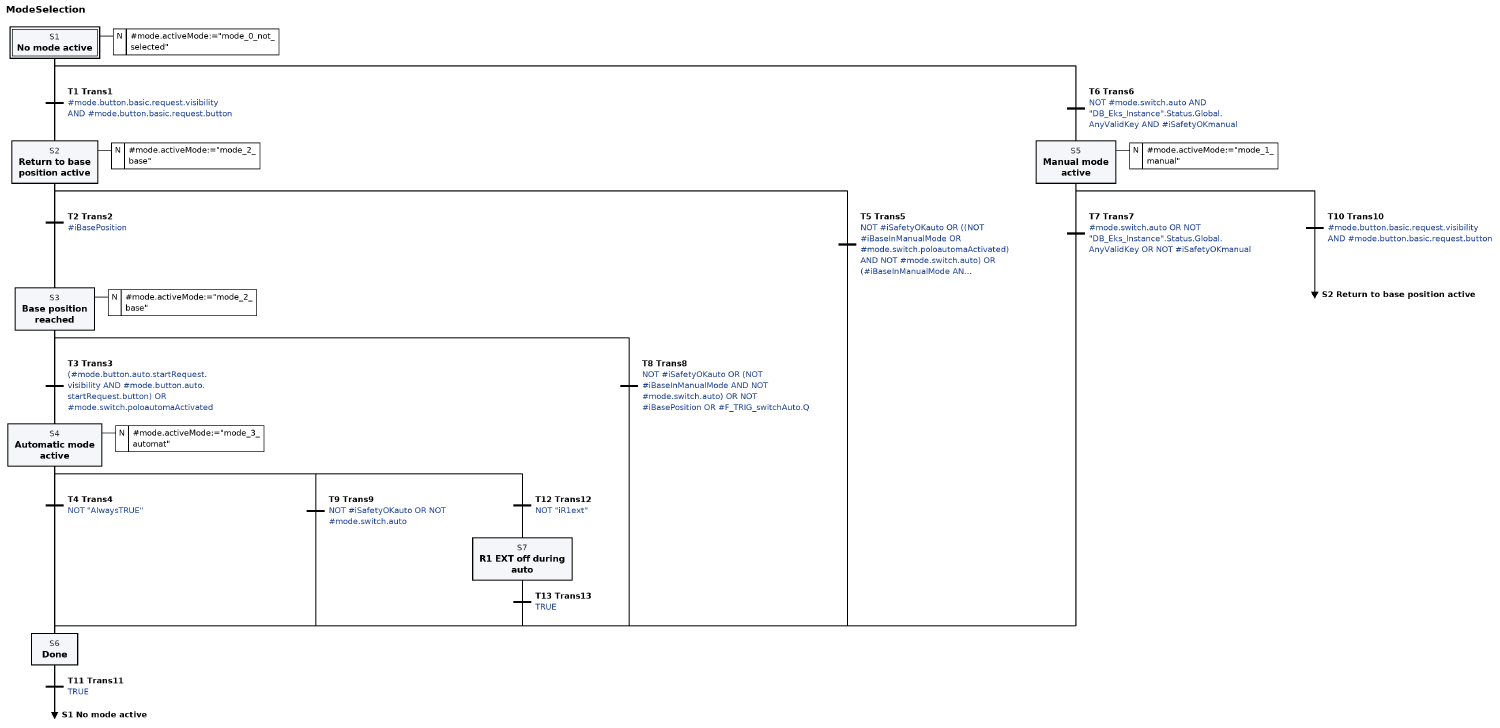
   // permanent pre-instructions
   NETWORK 1
   TITLE = mode init
      "ModeSelection_DB".mode.activeMode := "mode_0_not_selected";
   NETWORK 2
   TITLE = button visibility
      #mode.button.basic.request.visibility := #iSafetyOKauto AND ((#mode.switch.auto AND #"No mode active".X AND (NOT #iBaseInManualMode OR #mode.switch.poloautomaActivated)) OR (NOT #mode.switch.auto AND #"Manual mode active".X AND #iBaseInManualMode AND NOT #mode.switch.poloautomaActivated));
      #mode.button.auto.startRequest.visibility := #iSafetyOKauto AND #mode.switch.auto AND #"Base position reached".X AND NOT "SystemHMI".AlarmActive;
   NETWORK 3
   TITLE = semiauto switch off detection
      #F_TRIG_semiauto_switch(CLK := #mode.switch.poloautomaActivated);   // F_TRIG
   NETWORK 4
      #F_TRIG_switchAuto(CLK := #mode.switch.auto);   // F_TRIG

   // sequencer 1
   INITIAL_STEP "No mode active":   // S1, max time T#10S, warning time T#7S
              N    #mode.activeMode:="mode_0_not_selected"
   END_STEP
   TRANSITION Trans1 FROM "No mode active" TO "Return to base position active"   // T1
      := #mode.button.basic.request.visibility AND #mode.button.basic.request.button;
   END_TRANSITION
   TRANSITION Trans6 FROM "No mode active" TO "Manual mode active"   // T6
      := NOT #mode.switch.auto AND "DB_Eks_Instance".Status.Global.AnyValidKey AND #iSafetyOKmanual;
   END_TRANSITION
   STEP "Return to base position active":   // S2, max time T#10S, warning time T#7S
              N    #mode.activeMode:="mode_2_base"
   END_STEP
   TRANSITION Trans2 FROM "Return to base position active" TO "Base position reached"   // T2
      := #iBasePosition;
   END_TRANSITION
   TRANSITION Trans5 FROM "Return to base position active" TO Done   // T5
      := NOT #iSafetyOKauto OR ((NOT #iBaseInManualMode OR #mode.switch.poloautomaActivated) AND NOT #mode.switch.auto) OR (#iBaseInManualMode AND #mode.switch.auto AND NOT #mode.switch.poloautomaActivated) OR #F_TRIG_semiauto_switch.Q;
   END_TRANSITION
   STEP "Base position reached":   // S3, max time T#10S, warning time T#7S
              N    #mode.activeMode:="mode_2_base"
   END_STEP
   TRANSITION Trans3 FROM "Base position reached" TO "Automatic mode active"   // T3
      := (#mode.button.auto.startRequest.visibility AND #mode.button.auto.startRequest.button) OR #mode.switch.poloautomaActivated;
   END_TRANSITION
   TRANSITION Trans8 FROM "Base position reached" TO Done   // T8
      := NOT #iSafetyOKauto OR (NOT #iBaseInManualMode AND NOT #mode.switch.auto) OR NOT #iBasePosition OR #F_TRIG_switchAuto.Q;
   END_TRANSITION
   STEP "Automatic mode active":   // S4, max time T#10S, warning time T#7S
              N    #mode.activeMode:="mode_3_automat"
   END_STEP
   TRANSITION Trans4 FROM "Automatic mode active" TO Done   // T4
      := NOT "AlwaysTRUE";
   END_TRANSITION
   TRANSITION Trans9 FROM "Automatic mode active" TO Done   // T9
      := NOT #iSafetyOKauto OR NOT #mode.switch.auto;
   END_TRANSITION
   TRANSITION Trans12 FROM "Automatic mode active" TO "R1 EXT off during auto"   // T12
      := NOT "iR1ext";
   END_TRANSITION
   STEP "Manual mode active":   // S5, max time T#10S, warning time T#7S
              N    #mode.activeMode:="mode_1_manual"
   END_STEP
   TRANSITION Trans7 FROM "Manual mode active" TO Done   // T7
      := #mode.switch.auto OR NOT "DB_Eks_Instance".Status.Global.AnyValidKey OR NOT #iSafetyOKmanual;
   END_TRANSITION
   TRANSITION Trans10 FROM "Manual mode active" TO "Return to base position active"   // T10, jump
      := #mode.button.basic.request.visibility AND #mode.button.basic.request.button;
   END_TRANSITION
   STEP Done:   // S6, max time T#10S, warning time T#7S
   END_STEP
   TRANSITION Trans11 FROM Done TO "No mode active"   // T11, jump
      := TRUE;
   END_TRANSITION
   STEP "R1 EXT off during auto":   // S7, max time T#10S, warning time T#7S
   END_STEP
   TRANSITION Trans13 FROM "R1 EXT off during auto" TO Done   // T13
      := TRUE;
   END_TRANSITION

   // permanent post-instructions
   NETWORK 1
   TITLE = semiauto mode
      IF ((#mode.activeMode = "mode_2_base") OR (#mode.activeMode = "mode_3_automat")) AND #mode.switch.poloautomaActivated THEN
          #mode.activeMode := "mode_4_semiautomat";
      END_IF;
   NETWORK 2
   TITLE = previous mode
      #mode.modeChanged := #mode.activeMode <> #PrevMode;
      #PrevMode := #mode.activeMode;
END_FUNCTION_BLOCK

FUNCTION_BLOCK "Lamps"   // FB7, LAD
{ S7_Optimized_Access := 'TRUE' }
VERSION : 0.1
// stored: AutoNumber true, IsIECCheckEnabled false, IsRetainMemResEnabled false, MemoryReserve 100, SetENOAutomatically false, UDAEnableTagReadback false
   VAR
      R_TRIG_Instance { S7_SetPoint := 'True'} : R_TRIG;
      IEC_Timer_0_Instance { S7_SetPoint := 'True'} : TON_TIME;
   END_VAR
BEGIN

